   // GBK_TO_UNICODE[14568] := 16#AD6F;
   // GBK_TO_UNICODE[14569] := 16#74B7;
   // GBK_TO_UNICODE[14570] := 16#AD70;
   // GBK_TO_UNICODE[14571] := 16#74B8;
   // GBK_TO_UNICODE[14572] := 16#AD71;
   // GBK_TO_UNICODE[14573] := 16#74B9;
   // GBK_TO_UNICODE[14574] := 16#AD72;
   // GBK_TO_UNICODE[14575] := 16#74BB;
   // GBK_TO_UNICODE[14576] := 16#AD73;
   // GBK_TO_UNICODE[14577] := 16#74BC;
   // GBK_TO_UNICODE[14578] := 16#AD74;
   // GBK_TO_UNICODE[14579] := 16#74BD;
   // GBK_TO_UNICODE[14580] := 16#AD75;
   // GBK_TO_UNICODE[14581] := 16#74BE;
   // GBK_TO_UNICODE[14582] := 16#AD76;
   // GBK_TO_UNICODE[14583] := 16#74BF;
   // GBK_TO_UNICODE[14584] := 16#AD77;
   // GBK_TO_UNICODE[14585] := 16#74C0;
   // GBK_TO_UNICODE[14586] := 16#AD78;
   // GBK_TO_UNICODE[14587] := 16#74C1;
   // GBK_TO_UNICODE[14588] := 16#AD79;
   // GBK_TO_UNICODE[14589] := 16#74C2;
   // GBK_TO_UNICODE[14590] := 16#AD7A;
   // GBK_TO_UNICODE[14591] := 16#74C3;
   // GBK_TO_UNICODE[14592] := 16#AD7B;
   // GBK_TO_UNICODE[14593] := 16#74C4;
   // GBK_TO_UNICODE[14594] := 16#AD7C;
   // GBK_TO_UNICODE[14595] := 16#74C5;
   // GBK_TO_UNICODE[14596] := 16#AD7D;
   // GBK_TO_UNICODE[14597] := 16#74C6;
   // GBK_TO_UNICODE[14598] := 16#AD7E;
   // GBK_TO_UNICODE[14599] := 16#74C7;
   // GBK_TO_UNICODE[14600] := 16#AD80;
   // GBK_TO_UNICODE[14601] := 16#74C8;
   // GBK_TO_UNICODE[14602] := 16#AD81;
   // GBK_TO_UNICODE[14603] := 16#74C9;
   // GBK_TO_UNICODE[14604] := 16#AD82;
   // GBK_TO_UNICODE[14605] := 16#74CA;
   // GBK_TO_UNICODE[14606] := 16#AD83;
   // GBK_TO_UNICODE[14607] := 16#74CB;
   // GBK_TO_UNICODE[14608] := 16#AD84;
   // GBK_TO_UNICODE[14609] := 16#74CC;
   // GBK_TO_UNICODE[14610] := 16#AD85;
   // GBK_TO_UNICODE[14611] := 16#74CD;
   // GBK_TO_UNICODE[14612] := 16#AD86;
   // GBK_TO_UNICODE[14613] := 16#74CE;
   // GBK_TO_UNICODE[14614] := 16#AD87;
   // GBK_TO_UNICODE[14615] := 16#74CF;
   // GBK_TO_UNICODE[14616] := 16#AD88;
   // GBK_TO_UNICODE[14617] := 16#74D0;
   // GBK_TO_UNICODE[14618] := 16#AD89;
   // GBK_TO_UNICODE[14619] := 16#74D1;
   // GBK_TO_UNICODE[14620] := 16#AD8A;
   // GBK_TO_UNICODE[14621] := 16#74D3;
   // GBK_TO_UNICODE[14622] := 16#AD8B;
   // GBK_TO_UNICODE[14623] := 16#74D4;
   // GBK_TO_UNICODE[14624] := 16#AD8C;
   // GBK_TO_UNICODE[14625] := 16#74D5;
   // GBK_TO_UNICODE[14626] := 16#AD8D;
   // GBK_TO_UNICODE[14627] := 16#74D6;
   // GBK_TO_UNICODE[14628] := 16#AD8E;
   // GBK_TO_UNICODE[14629] := 16#74D7;
   // GBK_TO_UNICODE[14630] := 16#AD8F;
   // GBK_TO_UNICODE[14631] := 16#74D8;
   // GBK_TO_UNICODE[14632] := 16#AD90;
   // GBK_TO_UNICODE[14633] := 16#74D9;
   // GBK_TO_UNICODE[14634] := 16#AD91;
   // GBK_TO_UNICODE[14635] := 16#74DA;
   // GBK_TO_UNICODE[14636] := 16#AD92;
   // GBK_TO_UNICODE[14637] := 16#74DB;
   // GBK_TO_UNICODE[14638] := 16#AD93;
   // GBK_TO_UNICODE[14639] := 16#74DD;
   // GBK_TO_UNICODE[14640] := 16#AD94;
   // GBK_TO_UNICODE[14641] := 16#74DF;
   // GBK_TO_UNICODE[14642] := 16#AD95;
   // GBK_TO_UNICODE[14643] := 16#74E1;
   // GBK_TO_UNICODE[14644] := 16#AD96;
   // GBK_TO_UNICODE[14645] := 16#74E5;
   // GBK_TO_UNICODE[14646] := 16#AD97;
   // GBK_TO_UNICODE[14647] := 16#74E7;
   // GBK_TO_UNICODE[14648] := 16#AD98;
   // GBK_TO_UNICODE[14649] := 16#74E8;
   // GBK_TO_UNICODE[14650] := 16#AD99;
   // GBK_TO_UNICODE[14651] := 16#74E9;
   // GBK_TO_UNICODE[14652] := 16#AD9A;
   // GBK_TO_UNICODE[14653] := 16#74EA;
   // GBK_TO_UNICODE[14654] := 16#AD9B;
   // GBK_TO_UNICODE[14655] := 16#74EB;
   // GBK_TO_UNICODE[14656] := 16#AD9C;
   // GBK_TO_UNICODE[14657] := 16#74EC;
   // GBK_TO_UNICODE[14658] := 16#AD9D;
   // GBK_TO_UNICODE[14659] := 16#74ED;
   // GBK_TO_UNICODE[14660] := 16#AD9E;
   // GBK_TO_UNICODE[14661] := 16#74F0;
   // GBK_TO_UNICODE[14662] := 16#AD9F;
   // GBK_TO_UNICODE[14663] := 16#74F1;
   // GBK_TO_UNICODE[14664] := 16#ADA0;
   // GBK_TO_UNICODE[14665] := 16#74F2;
   // GBK_TO_UNICODE[14666] := 16#AE40;
   // GBK_TO_UNICODE[14667] := 16#74F3;
   // GBK_TO_UNICODE[14668] := 16#AE41;
   // GBK_TO_UNICODE[14669] := 16#74F5;
   // GBK_TO_UNICODE[14670] := 16#AE42;
   // GBK_TO_UNICODE[14671] := 16#74F8;
   // GBK_TO_UNICODE[14672] := 16#AE43;
   // GBK_TO_UNICODE[14673] := 16#74F9;
   // GBK_TO_UNICODE[14674] := 16#AE44;
   // GBK_TO_UNICODE[14675] := 16#74FA;
   // GBK_TO_UNICODE[14676] := 16#AE45;
   // GBK_TO_UNICODE[14677] := 16#74FB;
   // GBK_TO_UNICODE[14678] := 16#AE46;
   // GBK_TO_UNICODE[14679] := 16#74FC;
   // GBK_TO_UNICODE[14680] := 16#AE47;
   // GBK_TO_UNICODE[14681] := 16#74FD;
   // GBK_TO_UNICODE[14682] := 16#AE48;
   // GBK_TO_UNICODE[14683] := 16#74FE;
   // GBK_TO_UNICODE[14684] := 16#AE49;
   // GBK_TO_UNICODE[14685] := 16#7500;
   // GBK_TO_UNICODE[14686] := 16#AE4A;
   // GBK_TO_UNICODE[14687] := 16#7501;
   // GBK_TO_UNICODE[14688] := 16#AE4B;
   // GBK_TO_UNICODE[14689] := 16#7502;
   // GBK_TO_UNICODE[14690] := 16#AE4C;
   // GBK_TO_UNICODE[14691] := 16#7503;
   // GBK_TO_UNICODE[14692] := 16#AE4D;
   // GBK_TO_UNICODE[14693] := 16#7505;
   // GBK_TO_UNICODE[14694] := 16#AE4E;
   // GBK_TO_UNICODE[14695] := 16#7506;
   // GBK_TO_UNICODE[14696] := 16#AE4F;
   // GBK_TO_UNICODE[14697] := 16#7507;
   // GBK_TO_UNICODE[14698] := 16#AE50;
   // GBK_TO_UNICODE[14699] := 16#7508;
   // GBK_TO_UNICODE[14700] := 16#AE51;
   // GBK_TO_UNICODE[14701] := 16#7509;
   // GBK_TO_UNICODE[14702] := 16#AE52;
   // GBK_TO_UNICODE[14703] := 16#750A;
   // GBK_TO_UNICODE[14704] := 16#AE53;
   // GBK_TO_UNICODE[14705] := 16#750B;
   // GBK_TO_UNICODE[14706] := 16#AE54;
   // GBK_TO_UNICODE[14707] := 16#750C;
   // GBK_TO_UNICODE[14708] := 16#AE55;
   // GBK_TO_UNICODE[14709] := 16#750E;
   // GBK_TO_UNICODE[14710] := 16#AE56;
   // GBK_TO_UNICODE[14711] := 16#7510;
   // GBK_TO_UNICODE[14712] := 16#AE57;
   // GBK_TO_UNICODE[14713] := 16#7512;
   // GBK_TO_UNICODE[14714] := 16#AE58;
   // GBK_TO_UNICODE[14715] := 16#7514;
   // GBK_TO_UNICODE[14716] := 16#AE59;
   // GBK_TO_UNICODE[14717] := 16#7515;
   // GBK_TO_UNICODE[14718] := 16#AE5A;
   // GBK_TO_UNICODE[14719] := 16#7516;
   // GBK_TO_UNICODE[14720] := 16#AE5B;
   // GBK_TO_UNICODE[14721] := 16#7517;
   // GBK_TO_UNICODE[14722] := 16#AE5C;
   // GBK_TO_UNICODE[14723] := 16#751B;
   // GBK_TO_UNICODE[14724] := 16#AE5D;
   // GBK_TO_UNICODE[14725] := 16#751D;
   // GBK_TO_UNICODE[14726] := 16#AE5E;
   // GBK_TO_UNICODE[14727] := 16#751E;
   // GBK_TO_UNICODE[14728] := 16#AE5F;
   // GBK_TO_UNICODE[14729] := 16#7520;
   // GBK_TO_UNICODE[14730] := 16#AE60;
   // GBK_TO_UNICODE[14731] := 16#7521;
   // GBK_TO_UNICODE[14732] := 16#AE61;
   // GBK_TO_UNICODE[14733] := 16#7522;
   // GBK_TO_UNICODE[14734] := 16#AE62;
   // GBK_TO_UNICODE[14735] := 16#7523;
   // GBK_TO_UNICODE[14736] := 16#AE63;
   // GBK_TO_UNICODE[14737] := 16#7524;
   // GBK_TO_UNICODE[14738] := 16#AE64;
   // GBK_TO_UNICODE[14739] := 16#7526;
   // GBK_TO_UNICODE[14740] := 16#AE65;
   // GBK_TO_UNICODE[14741] := 16#7527;
   // GBK_TO_UNICODE[14742] := 16#AE66;
   // GBK_TO_UNICODE[14743] := 16#752A;
   // GBK_TO_UNICODE[14744] := 16#AE67;
   // GBK_TO_UNICODE[14745] := 16#752E;
   // GBK_TO_UNICODE[14746] := 16#AE68;
   // GBK_TO_UNICODE[14747] := 16#7534;
   // GBK_TO_UNICODE[14748] := 16#AE69;
   // GBK_TO_UNICODE[14749] := 16#7536;
   // GBK_TO_UNICODE[14750] := 16#AE6A;
   // GBK_TO_UNICODE[14751] := 16#7539;
   // GBK_TO_UNICODE[14752] := 16#AE6B;
   // GBK_TO_UNICODE[14753] := 16#753C;
   // GBK_TO_UNICODE[14754] := 16#AE6C;
   // GBK_TO_UNICODE[14755] := 16#753D;
   // GBK_TO_UNICODE[14756] := 16#AE6D;
   // GBK_TO_UNICODE[14757] := 16#753F;
   // GBK_TO_UNICODE[14758] := 16#AE6E;
   // GBK_TO_UNICODE[14759] := 16#7541;
   // GBK_TO_UNICODE[14760] := 16#AE6F;
   // GBK_TO_UNICODE[14761] := 16#7542;
   // GBK_TO_UNICODE[14762] := 16#AE70;
   // GBK_TO_UNICODE[14763] := 16#7543;
   // GBK_TO_UNICODE[14764] := 16#AE71;
   // GBK_TO_UNICODE[14765] := 16#7544;
   // GBK_TO_UNICODE[14766] := 16#AE72;
   // GBK_TO_UNICODE[14767] := 16#7546;
   // GBK_TO_UNICODE[14768] := 16#AE73;
   // GBK_TO_UNICODE[14769] := 16#7547;
   // GBK_TO_UNICODE[14770] := 16#AE74;
   // GBK_TO_UNICODE[14771] := 16#7549;
   // GBK_TO_UNICODE[14772] := 16#AE75;
   // GBK_TO_UNICODE[14773] := 16#754A;
   // GBK_TO_UNICODE[14774] := 16#AE76;
   // GBK_TO_UNICODE[14775] := 16#754D;
   // GBK_TO_UNICODE[14776] := 16#AE77;
   // GBK_TO_UNICODE[14777] := 16#7550;
   // GBK_TO_UNICODE[14778] := 16#AE78;
   // GBK_TO_UNICODE[14779] := 16#7551;
   // GBK_TO_UNICODE[14780] := 16#AE79;
   // GBK_TO_UNICODE[14781] := 16#7552;
   // GBK_TO_UNICODE[14782] := 16#AE7A;
   // GBK_TO_UNICODE[14783] := 16#7553;
   // GBK_TO_UNICODE[14784] := 16#AE7B;
   // GBK_TO_UNICODE[14785] := 16#7555;
   // GBK_TO_UNICODE[14786] := 16#AE7C;
   // GBK_TO_UNICODE[14787] := 16#7556;
   // GBK_TO_UNICODE[14788] := 16#AE7D;
   // GBK_TO_UNICODE[14789] := 16#7557;
   // GBK_TO_UNICODE[14790] := 16#AE7E;
   // GBK_TO_UNICODE[14791] := 16#7558;
   // GBK_TO_UNICODE[14792] := 16#AE80;
   // GBK_TO_UNICODE[14793] := 16#755D;
   // GBK_TO_UNICODE[14794] := 16#AE81;
   // GBK_TO_UNICODE[14795] := 16#755E;
   // GBK_TO_UNICODE[14796] := 16#AE82;
   // GBK_TO_UNICODE[14797] := 16#755F;
   // GBK_TO_UNICODE[14798] := 16#AE83;
   // GBK_TO_UNICODE[14799] := 16#7560;
   // GBK_TO_UNICODE[14800] := 16#AE84;
   // GBK_TO_UNICODE[14801] := 16#7561;
   // GBK_TO_UNICODE[14802] := 16#AE85;
   // GBK_TO_UNICODE[14803] := 16#7562;
   // GBK_TO_UNICODE[14804] := 16#AE86;
   // GBK_TO_UNICODE[14805] := 16#7563;
   // GBK_TO_UNICODE[14806] := 16#AE87;
   // GBK_TO_UNICODE[14807] := 16#7564;
   // GBK_TO_UNICODE[14808] := 16#AE88;
   // GBK_TO_UNICODE[14809] := 16#7567;
   // GBK_TO_UNICODE[14810] := 16#AE89;
   // GBK_TO_UNICODE[14811] := 16#7568;
   // GBK_TO_UNICODE[14812] := 16#AE8A;
   // GBK_TO_UNICODE[14813] := 16#7569;
   // GBK_TO_UNICODE[14814] := 16#AE8B;
   // GBK_TO_UNICODE[14815] := 16#756B;
   // GBK_TO_UNICODE[14816] := 16#AE8C;
   // GBK_TO_UNICODE[14817] := 16#756C;
   // GBK_TO_UNICODE[14818] := 16#AE8D;
   // GBK_TO_UNICODE[14819] := 16#756D;
   // GBK_TO_UNICODE[14820] := 16#AE8E;
   // GBK_TO_UNICODE[14821] := 16#756E;
   // GBK_TO_UNICODE[14822] := 16#AE8F;
   // GBK_TO_UNICODE[14823] := 16#756F;
   // GBK_TO_UNICODE[14824] := 16#AE90;
   // GBK_TO_UNICODE[14825] := 16#7570;
   // GBK_TO_UNICODE[14826] := 16#AE91;
   // GBK_TO_UNICODE[14827] := 16#7571;
   // GBK_TO_UNICODE[14828] := 16#AE92;
   // GBK_TO_UNICODE[14829] := 16#7573;
   // GBK_TO_UNICODE[14830] := 16#AE93;
   // GBK_TO_UNICODE[14831] := 16#7575;
   // GBK_TO_UNICODE[14832] := 16#AE94;
   // GBK_TO_UNICODE[14833] := 16#7576;
   // GBK_TO_UNICODE[14834] := 16#AE95;
   // GBK_TO_UNICODE[14835] := 16#7577;
   // GBK_TO_UNICODE[14836] := 16#AE96;
   // GBK_TO_UNICODE[14837] := 16#757A;
   // GBK_TO_UNICODE[14838] := 16#AE97;
   // GBK_TO_UNICODE[14839] := 16#757B;
   // GBK_TO_UNICODE[14840] := 16#AE98;
   // GBK_TO_UNICODE[14841] := 16#757C;
   // GBK_TO_UNICODE[14842] := 16#AE99;
   // GBK_TO_UNICODE[14843] := 16#757D;
   // GBK_TO_UNICODE[14844] := 16#AE9A;
   // GBK_TO_UNICODE[14845] := 16#757E;
   // GBK_TO_UNICODE[14846] := 16#AE9B;
   // GBK_TO_UNICODE[14847] := 16#7580;
   // GBK_TO_UNICODE[14848] := 16#AE9C;
   // GBK_TO_UNICODE[14849] := 16#7581;
   // GBK_TO_UNICODE[14850] := 16#AE9D;
   // GBK_TO_UNICODE[14851] := 16#7582;
   // GBK_TO_UNICODE[14852] := 16#AE9E;
   // GBK_TO_UNICODE[14853] := 16#7584;
   // GBK_TO_UNICODE[14854] := 16#AE9F;
   // GBK_TO_UNICODE[14855] := 16#7585;
   // GBK_TO_UNICODE[14856] := 16#AEA0;
   // GBK_TO_UNICODE[14857] := 16#7587;
   // GBK_TO_UNICODE[14858] := 16#AF40;
   // GBK_TO_UNICODE[14859] := 16#7588;
   // GBK_TO_UNICODE[14860] := 16#AF41;
   // GBK_TO_UNICODE[14861] := 16#7589;
   // GBK_TO_UNICODE[14862] := 16#AF42;
   // GBK_TO_UNICODE[14863] := 16#758A;
   // GBK_TO_UNICODE[14864] := 16#AF43;
   // GBK_TO_UNICODE[14865] := 16#758C;
   // GBK_TO_UNICODE[14866] := 16#AF44;
   // GBK_TO_UNICODE[14867] := 16#758D;
   // GBK_TO_UNICODE[14868] := 16#AF45;
   // GBK_TO_UNICODE[14869] := 16#758E;
   // GBK_TO_UNICODE[14870] := 16#AF46;
   // GBK_TO_UNICODE[14871] := 16#7590;
   // GBK_TO_UNICODE[14872] := 16#AF47;
   // GBK_TO_UNICODE[14873] := 16#7593;
   // GBK_TO_UNICODE[14874] := 16#AF48;
   // GBK_TO_UNICODE[14875] := 16#7595;
   // GBK_TO_UNICODE[14876] := 16#AF49;
   // GBK_TO_UNICODE[14877] := 16#7598;
   // GBK_TO_UNICODE[14878] := 16#AF4A;
   // GBK_TO_UNICODE[14879] := 16#759B;
   // GBK_TO_UNICODE[14880] := 16#AF4B;
   // GBK_TO_UNICODE[14881] := 16#759C;
   // GBK_TO_UNICODE[14882] := 16#AF4C;
   // GBK_TO_UNICODE[14883] := 16#759E;
   // GBK_TO_UNICODE[14884] := 16#AF4D;
   // GBK_TO_UNICODE[14885] := 16#75A2;
   // GBK_TO_UNICODE[14886] := 16#AF4E;
   // GBK_TO_UNICODE[14887] := 16#75A6;
   // GBK_TO_UNICODE[14888] := 16#AF4F;
   // GBK_TO_UNICODE[14889] := 16#75A7;
   // GBK_TO_UNICODE[14890] := 16#AF50;
   // GBK_TO_UNICODE[14891] := 16#75A8;
   // GBK_TO_UNICODE[14892] := 16#AF51;
   // GBK_TO_UNICODE[14893] := 16#75A9;
   // GBK_TO_UNICODE[14894] := 16#AF52;
   // GBK_TO_UNICODE[14895] := 16#75AA;
   // GBK_TO_UNICODE[14896] := 16#AF53;
   // GBK_TO_UNICODE[14897] := 16#75AD;
   // GBK_TO_UNICODE[14898] := 16#AF54;
   // GBK_TO_UNICODE[14899] := 16#75B6;
   // GBK_TO_UNICODE[14900] := 16#AF55;
   // GBK_TO_UNICODE[14901] := 16#75B7;
   // GBK_TO_UNICODE[14902] := 16#AF56;
   // GBK_TO_UNICODE[14903] := 16#75BA;
   // GBK_TO_UNICODE[14904] := 16#AF57;
   // GBK_TO_UNICODE[14905] := 16#75BB;
   // GBK_TO_UNICODE[14906] := 16#AF58;
   // GBK_TO_UNICODE[14907] := 16#75BF;
   // GBK_TO_UNICODE[14908] := 16#AF59;
   // GBK_TO_UNICODE[14909] := 16#75C0;
   // GBK_TO_UNICODE[14910] := 16#AF5A;
   // GBK_TO_UNICODE[14911] := 16#75C1;
   // GBK_TO_UNICODE[14912] := 16#AF5B;
   // GBK_TO_UNICODE[14913] := 16#75C6;
   // GBK_TO_UNICODE[14914] := 16#AF5C;
   // GBK_TO_UNICODE[14915] := 16#75CB;
   // GBK_TO_UNICODE[14916] := 16#AF5D;
   // GBK_TO_UNICODE[14917] := 16#75CC;
   // GBK_TO_UNICODE[14918] := 16#AF5E;
   // GBK_TO_UNICODE[14919] := 16#75CE;
   // GBK_TO_UNICODE[14920] := 16#AF5F;
   // GBK_TO_UNICODE[14921] := 16#75CF;
   // GBK_TO_UNICODE[14922] := 16#AF60;
   // GBK_TO_UNICODE[14923] := 16#75D0;
   // GBK_TO_UNICODE[14924] := 16#AF61;
   // GBK_TO_UNICODE[14925] := 16#75D1;
   // GBK_TO_UNICODE[14926] := 16#AF62;
   // GBK_TO_UNICODE[14927] := 16#75D3;
   // GBK_TO_UNICODE[14928] := 16#AF63;
   // GBK_TO_UNICODE[14929] := 16#75D7;
   // GBK_TO_UNICODE[14930] := 16#AF64;
   // GBK_TO_UNICODE[14931] := 16#75D9;
   // GBK_TO_UNICODE[14932] := 16#AF65;
   // GBK_TO_UNICODE[14933] := 16#75DA;
   // GBK_TO_UNICODE[14934] := 16#AF66;
   // GBK_TO_UNICODE[14935] := 16#75DC;
   // GBK_TO_UNICODE[14936] := 16#AF67;
   // GBK_TO_UNICODE[14937] := 16#75DD;
   // GBK_TO_UNICODE[14938] := 16#AF68;
   // GBK_TO_UNICODE[14939] := 16#75DF;
   // GBK_TO_UNICODE[14940] := 16#AF69;
   // GBK_TO_UNICODE[14941] := 16#75E0;
   // GBK_TO_UNICODE[14942] := 16#AF6A;
   // GBK_TO_UNICODE[14943] := 16#75E1;
   // GBK_TO_UNICODE[14944] := 16#AF6B;
   // GBK_TO_UNICODE[14945] := 16#75E5;
   // GBK_TO_UNICODE[14946] := 16#AF6C;
   // GBK_TO_UNICODE[14947] := 16#75E9;
   // GBK_TO_UNICODE[14948] := 16#AF6D;
   // GBK_TO_UNICODE[14949] := 16#75EC;
   // GBK_TO_UNICODE[14950] := 16#AF6E;
   // GBK_TO_UNICODE[14951] := 16#75ED;
   // GBK_TO_UNICODE[14952] := 16#AF6F;
   // GBK_TO_UNICODE[14953] := 16#75EE;
   // GBK_TO_UNICODE[14954] := 16#AF70;
   // GBK_TO_UNICODE[14955] := 16#75EF;
   // GBK_TO_UNICODE[14956] := 16#AF71;
   // GBK_TO_UNICODE[14957] := 16#75F2;
   // GBK_TO_UNICODE[14958] := 16#AF72;
   // GBK_TO_UNICODE[14959] := 16#75F3;
   // GBK_TO_UNICODE[14960] := 16#AF73;
   // GBK_TO_UNICODE[14961] := 16#75F5;
   // GBK_TO_UNICODE[14962] := 16#AF74;
   // GBK_TO_UNICODE[14963] := 16#75F6;
   // GBK_TO_UNICODE[14964] := 16#AF75;
   // GBK_TO_UNICODE[14965] := 16#75F7;
   // GBK_TO_UNICODE[14966] := 16#AF76;
   // GBK_TO_UNICODE[14967] := 16#75F8;
   // GBK_TO_UNICODE[14968] := 16#AF77;
   // GBK_TO_UNICODE[14969] := 16#75FA;
   // GBK_TO_UNICODE[14970] := 16#AF78;
   // GBK_TO_UNICODE[14971] := 16#75FB;
   // GBK_TO_UNICODE[14972] := 16#AF79;
   // GBK_TO_UNICODE[14973] := 16#75FD;
   // GBK_TO_UNICODE[14974] := 16#AF7A;
   // GBK_TO_UNICODE[14975] := 16#75FE;
   // GBK_TO_UNICODE[14976] := 16#AF7B;
   // GBK_TO_UNICODE[14977] := 16#7602;
   // GBK_TO_UNICODE[14978] := 16#AF7C;
   // GBK_TO_UNICODE[14979] := 16#7604;
   // GBK_TO_UNICODE[14980] := 16#AF7D;
   // GBK_TO_UNICODE[14981] := 16#7606;
   // GBK_TO_UNICODE[14982] := 16#AF7E;
   // GBK_TO_UNICODE[14983] := 16#7607;
   // GBK_TO_UNICODE[14984] := 16#AF80;
   // GBK_TO_UNICODE[14985] := 16#7608;
   // GBK_TO_UNICODE[14986] := 16#AF81;
   // GBK_TO_UNICODE[14987] := 16#7609;
   // GBK_TO_UNICODE[14988] := 16#AF82;
   // GBK_TO_UNICODE[14989] := 16#760B;
   // GBK_TO_UNICODE[14990] := 16#AF83;
   // GBK_TO_UNICODE[14991] := 16#760D;
   // GBK_TO_UNICODE[14992] := 16#AF84;
   // GBK_TO_UNICODE[14993] := 16#760E;
   // GBK_TO_UNICODE[14994] := 16#AF85;
   // GBK_TO_UNICODE[14995] := 16#760F;
   // GBK_TO_UNICODE[14996] := 16#AF86;
   // GBK_TO_UNICODE[14997] := 16#7611;
   // GBK_TO_UNICODE[14998] := 16#AF87;
   // GBK_TO_UNICODE[14999] := 16#7612;
   // GBK_TO_UNICODE[15000] := 16#AF88;
   // GBK_TO_UNICODE[15001] := 16#7613;
   // GBK_TO_UNICODE[15002] := 16#AF89;
   // GBK_TO_UNICODE[15003] := 16#7614;
   // GBK_TO_UNICODE[15004] := 16#AF8A;
   // GBK_TO_UNICODE[15005] := 16#7616;
   // GBK_TO_UNICODE[15006] := 16#AF8B;
   // GBK_TO_UNICODE[15007] := 16#761A;
   // GBK_TO_UNICODE[15008] := 16#AF8C;
   // GBK_TO_UNICODE[15009] := 16#761C;
   // GBK_TO_UNICODE[15010] := 16#AF8D;
   // GBK_TO_UNICODE[15011] := 16#761D;
   // GBK_TO_UNICODE[15012] := 16#AF8E;
   // GBK_TO_UNICODE[15013] := 16#761E;
   // GBK_TO_UNICODE[15014] := 16#AF8F;
   // GBK_TO_UNICODE[15015] := 16#7621;
   // GBK_TO_UNICODE[15016] := 16#AF90;
   // GBK_TO_UNICODE[15017] := 16#7623;
   // GBK_TO_UNICODE[15018] := 16#AF91;
   // GBK_TO_UNICODE[15019] := 16#7627;
   // GBK_TO_UNICODE[15020] := 16#AF92;
   // GBK_TO_UNICODE[15021] := 16#7628;
   // GBK_TO_UNICODE[15022] := 16#AF93;
   // GBK_TO_UNICODE[15023] := 16#762C;
   // GBK_TO_UNICODE[15024] := 16#AF94;
   // GBK_TO_UNICODE[15025] := 16#762E;
   // GBK_TO_UNICODE[15026] := 16#AF95;
   // GBK_TO_UNICODE[15027] := 16#762F;
   // GBK_TO_UNICODE[15028] := 16#AF96;
   // GBK_TO_UNICODE[15029] := 16#7631;
   // GBK_TO_UNICODE[15030] := 16#AF97;
   // GBK_TO_UNICODE[15031] := 16#7632;
   // GBK_TO_UNICODE[15032] := 16#AF98;
   // GBK_TO_UNICODE[15033] := 16#7636;
   // GBK_TO_UNICODE[15034] := 16#AF99;
   // GBK_TO_UNICODE[15035] := 16#7637;
   // GBK_TO_UNICODE[15036] := 16#AF9A;
   // GBK_TO_UNICODE[15037] := 16#7639;
   // GBK_TO_UNICODE[15038] := 16#AF9B;
   // GBK_TO_UNICODE[15039] := 16#763A;
   // GBK_TO_UNICODE[15040] := 16#AF9C;
   // GBK_TO_UNICODE[15041] := 16#763B;
   // GBK_TO_UNICODE[15042] := 16#AF9D;
   // GBK_TO_UNICODE[15043] := 16#763D;
   // GBK_TO_UNICODE[15044] := 16#AF9E;
   // GBK_TO_UNICODE[15045] := 16#7641;
   // GBK_TO_UNICODE[15046] := 16#AF9F;
   // GBK_TO_UNICODE[15047] := 16#7642;
   // GBK_TO_UNICODE[15048] := 16#AFA0;
   // GBK_TO_UNICODE[15049] := 16#7644;
   // GBK_TO_UNICODE[15050] := 16#B040;
   // GBK_TO_UNICODE[15051] := 16#7645;
   // GBK_TO_UNICODE[15052] := 16#B041;
   // GBK_TO_UNICODE[15053] := 16#7646;
   // GBK_TO_UNICODE[15054] := 16#B042;
   // GBK_TO_UNICODE[15055] := 16#7647;
   // GBK_TO_UNICODE[15056] := 16#B043;
   // GBK_TO_UNICODE[15057] := 16#7648;
   // GBK_TO_UNICODE[15058] := 16#B044;
   // GBK_TO_UNICODE[15059] := 16#7649;
   // GBK_TO_UNICODE[15060] := 16#B045;
   // GBK_TO_UNICODE[15061] := 16#764A;
   // GBK_TO_UNICODE[15062] := 16#B046;
   // GBK_TO_UNICODE[15063] := 16#764B;
   // GBK_TO_UNICODE[15064] := 16#B047;
   // GBK_TO_UNICODE[15065] := 16#764E;
   // GBK_TO_UNICODE[15066] := 16#B048;
   // GBK_TO_UNICODE[15067] := 16#764F;
   // GBK_TO_UNICODE[15068] := 16#B049;
   // GBK_TO_UNICODE[15069] := 16#7650;
   // GBK_TO_UNICODE[15070] := 16#B04A;
   // GBK_TO_UNICODE[15071] := 16#7651;
   // GBK_TO_UNICODE[15072] := 16#B04B;
   // GBK_TO_UNICODE[15073] := 16#7652;
   // GBK_TO_UNICODE[15074] := 16#B04C;
   // GBK_TO_UNICODE[15075] := 16#7653;
   // GBK_TO_UNICODE[15076] := 16#B04D;
   // GBK_TO_UNICODE[15077] := 16#7655;
   // GBK_TO_UNICODE[15078] := 16#B04E;
   // GBK_TO_UNICODE[15079] := 16#7657;
   // GBK_TO_UNICODE[15080] := 16#B04F;
   // GBK_TO_UNICODE[15081] := 16#7658;
   // GBK_TO_UNICODE[15082] := 16#B050;
   // GBK_TO_UNICODE[15083] := 16#7659;
   // GBK_TO_UNICODE[15084] := 16#B051;
   // GBK_TO_UNICODE[15085] := 16#765A;
   // GBK_TO_UNICODE[15086] := 16#B052;
   // GBK_TO_UNICODE[15087] := 16#765B;
   // GBK_TO_UNICODE[15088] := 16#B053;
   // GBK_TO_UNICODE[15089] := 16#765D;
   // GBK_TO_UNICODE[15090] := 16#B054;
   // GBK_TO_UNICODE[15091] := 16#765F;
   // GBK_TO_UNICODE[15092] := 16#B055;
   // GBK_TO_UNICODE[15093] := 16#7660;
   // GBK_TO_UNICODE[15094] := 16#B056;
   // GBK_TO_UNICODE[15095] := 16#7661;
   // GBK_TO_UNICODE[15096] := 16#B057;
   // GBK_TO_UNICODE[15097] := 16#7662;
   // GBK_TO_UNICODE[15098] := 16#B058;
   // GBK_TO_UNICODE[15099] := 16#7664;
   // GBK_TO_UNICODE[15100] := 16#B059;
   // GBK_TO_UNICODE[15101] := 16#7665;
   // GBK_TO_UNICODE[15102] := 16#B05A;
   // GBK_TO_UNICODE[15103] := 16#7666;
   // GBK_TO_UNICODE[15104] := 16#B05B;
   // GBK_TO_UNICODE[15105] := 16#7667;
   // GBK_TO_UNICODE[15106] := 16#B05C;
   // GBK_TO_UNICODE[15107] := 16#7668;
   // GBK_TO_UNICODE[15108] := 16#B05D;
   // GBK_TO_UNICODE[15109] := 16#7669;
   // GBK_TO_UNICODE[15110] := 16#B05E;
   // GBK_TO_UNICODE[15111] := 16#766A;
   // GBK_TO_UNICODE[15112] := 16#B05F;
   // GBK_TO_UNICODE[15113] := 16#766C;
   // GBK_TO_UNICODE[15114] := 16#B060;
   // GBK_TO_UNICODE[15115] := 16#766D;
   // GBK_TO_UNICODE[15116] := 16#B061;
   // GBK_TO_UNICODE[15117] := 16#766E;
   // GBK_TO_UNICODE[15118] := 16#B062;
   // GBK_TO_UNICODE[15119] := 16#7670;
   // GBK_TO_UNICODE[15120] := 16#B063;
   // GBK_TO_UNICODE[15121] := 16#7671;
   // GBK_TO_UNICODE[15122] := 16#B064;
   // GBK_TO_UNICODE[15123] := 16#7672;
   // GBK_TO_UNICODE[15124] := 16#B065;
   // GBK_TO_UNICODE[15125] := 16#7673;
   // GBK_TO_UNICODE[15126] := 16#B066;
   // GBK_TO_UNICODE[15127] := 16#7674;
   // GBK_TO_UNICODE[15128] := 16#B067;
   // GBK_TO_UNICODE[15129] := 16#7675;
   // GBK_TO_UNICODE[15130] := 16#B068;
   // GBK_TO_UNICODE[15131] := 16#7676;
   // GBK_TO_UNICODE[15132] := 16#B069;
   // GBK_TO_UNICODE[15133] := 16#7677;
   // GBK_TO_UNICODE[15134] := 16#B06A;
   // GBK_TO_UNICODE[15135] := 16#7679;
   // GBK_TO_UNICODE[15136] := 16#B06B;
   // GBK_TO_UNICODE[15137] := 16#767A;
   // GBK_TO_UNICODE[15138] := 16#B06C;
   // GBK_TO_UNICODE[15139] := 16#767C;
   // GBK_TO_UNICODE[15140] := 16#B06D;
   // GBK_TO_UNICODE[15141] := 16#767F;
   // GBK_TO_UNICODE[15142] := 16#B06E;
   // GBK_TO_UNICODE[15143] := 16#7680;
   // GBK_TO_UNICODE[15144] := 16#B06F;
   // GBK_TO_UNICODE[15145] := 16#7681;
   // GBK_TO_UNICODE[15146] := 16#B070;
   // GBK_TO_UNICODE[15147] := 16#7683;
   // GBK_TO_UNICODE[15148] := 16#B071;
   // GBK_TO_UNICODE[15149] := 16#7685;
   // GBK_TO_UNICODE[15150] := 16#B072;
   // GBK_TO_UNICODE[15151] := 16#7689;
   // GBK_TO_UNICODE[15152] := 16#B073;
   // GBK_TO_UNICODE[15153] := 16#768A;
   // GBK_TO_UNICODE[15154] := 16#B074;
   // GBK_TO_UNICODE[15155] := 16#768C;
   // GBK_TO_UNICODE[15156] := 16#B075;
   // GBK_TO_UNICODE[15157] := 16#768D;
   // GBK_TO_UNICODE[15158] := 16#B076;
   // GBK_TO_UNICODE[15159] := 16#768F;
   // GBK_TO_UNICODE[15160] := 16#B077;
   // GBK_TO_UNICODE[15161] := 16#7690;
   // GBK_TO_UNICODE[15162] := 16#B078;
   // GBK_TO_UNICODE[15163] := 16#7692;
   // GBK_TO_UNICODE[15164] := 16#B079;
   // GBK_TO_UNICODE[15165] := 16#7694;
   // GBK_TO_UNICODE[15166] := 16#B07A;
   // GBK_TO_UNICODE[15167] := 16#7695;
   // GBK_TO_UNICODE[15168] := 16#B07B;
   // GBK_TO_UNICODE[15169] := 16#7697;
   // GBK_TO_UNICODE[15170] := 16#B07C;
   // GBK_TO_UNICODE[15171] := 16#7698;
   // GBK_TO_UNICODE[15172] := 16#B07D;
   // GBK_TO_UNICODE[15173] := 16#769A;
   // GBK_TO_UNICODE[15174] := 16#B07E;
   // GBK_TO_UNICODE[15175] := 16#769B;
   // GBK_TO_UNICODE[15176] := 16#B080;
   // GBK_TO_UNICODE[15177] := 16#769C;
   // GBK_TO_UNICODE[15178] := 16#B081;
   // GBK_TO_UNICODE[15179] := 16#769D;
   // GBK_TO_UNICODE[15180] := 16#B082;
   // GBK_TO_UNICODE[15181] := 16#769E;
   // GBK_TO_UNICODE[15182] := 16#B083;
   // GBK_TO_UNICODE[15183] := 16#769F;
   // GBK_TO_UNICODE[15184] := 16#B084;
   // GBK_TO_UNICODE[15185] := 16#76A0;
   // GBK_TO_UNICODE[15186] := 16#B085;
   // GBK_TO_UNICODE[15187] := 16#76A1;
   // GBK_TO_UNICODE[15188] := 16#B086;
   // GBK_TO_UNICODE[15189] := 16#76A2;
   // GBK_TO_UNICODE[15190] := 16#B087;
   // GBK_TO_UNICODE[15191] := 16#76A3;
   // GBK_TO_UNICODE[15192] := 16#B088;
   // GBK_TO_UNICODE[15193] := 16#76A5;
   // GBK_TO_UNICODE[15194] := 16#B089;
   // GBK_TO_UNICODE[15195] := 16#76A6;
   // GBK_TO_UNICODE[15196] := 16#B08A;
   // GBK_TO_UNICODE[15197] := 16#76A7;
   // GBK_TO_UNICODE[15198] := 16#B08B;
   // GBK_TO_UNICODE[15199] := 16#76A8;
   // GBK_TO_UNICODE[15200] := 16#B08C;
   // GBK_TO_UNICODE[15201] := 16#76A9;
   // GBK_TO_UNICODE[15202] := 16#B08D;
   // GBK_TO_UNICODE[15203] := 16#76AA;
   // GBK_TO_UNICODE[15204] := 16#B08E;
   // GBK_TO_UNICODE[15205] := 16#76AB;
   // GBK_TO_UNICODE[15206] := 16#B08F;
   // GBK_TO_UNICODE[15207] := 16#76AC;
   // GBK_TO_UNICODE[15208] := 16#B090;
   // GBK_TO_UNICODE[15209] := 16#76AD;
   // GBK_TO_UNICODE[15210] := 16#B091;
   // GBK_TO_UNICODE[15211] := 16#76AF;
   // GBK_TO_UNICODE[15212] := 16#B092;
   // GBK_TO_UNICODE[15213] := 16#76B0;
   // GBK_TO_UNICODE[15214] := 16#B093;
   // GBK_TO_UNICODE[15215] := 16#76B3;
   // GBK_TO_UNICODE[15216] := 16#B094;
   // GBK_TO_UNICODE[15217] := 16#76B5;
   // GBK_TO_UNICODE[15218] := 16#B095;
   // GBK_TO_UNICODE[15219] := 16#76B6;
   // GBK_TO_UNICODE[15220] := 16#B096;
   // GBK_TO_UNICODE[15221] := 16#76B7;
   // GBK_TO_UNICODE[15222] := 16#B097;
   // GBK_TO_UNICODE[15223] := 16#76B8;
   // GBK_TO_UNICODE[15224] := 16#B098;
   // GBK_TO_UNICODE[15225] := 16#76B9;
   // GBK_TO_UNICODE[15226] := 16#B099;
   // GBK_TO_UNICODE[15227] := 16#76BA;
   // GBK_TO_UNICODE[15228] := 16#B09A;
   // GBK_TO_UNICODE[15229] := 16#76BB;
   // GBK_TO_UNICODE[15230] := 16#B09B;
   // GBK_TO_UNICODE[15231] := 16#76BC;
   // GBK_TO_UNICODE[15232] := 16#B09C;
   // GBK_TO_UNICODE[15233] := 16#76BD;
   // GBK_TO_UNICODE[15234] := 16#B09D;
   // GBK_TO_UNICODE[15235] := 16#76BE;
   // GBK_TO_UNICODE[15236] := 16#B09E;
   // GBK_TO_UNICODE[15237] := 16#76C0;
   // GBK_TO_UNICODE[15238] := 16#B09F;
   // GBK_TO_UNICODE[15239] := 16#76C1;
   // GBK_TO_UNICODE[15240] := 16#B0A0;
   // GBK_TO_UNICODE[15241] := 16#76C3;
   // GBK_TO_UNICODE[15242] := 16#B0A1;
   // GBK_TO_UNICODE[15243] := 16#554A;
   // GBK_TO_UNICODE[15244] := 16#B0A2;
   // GBK_TO_UNICODE[15245] := 16#963F;
   // GBK_TO_UNICODE[15246] := 16#B0A3;
   // GBK_TO_UNICODE[15247] := 16#57C3;
   // GBK_TO_UNICODE[15248] := 16#B0A4;
   // GBK_TO_UNICODE[15249] := 16#6328;
   // GBK_TO_UNICODE[15250] := 16#B0A5;
   // GBK_TO_UNICODE[15251] := 16#54CE;
   // GBK_TO_UNICODE[15252] := 16#B0A6;
   // GBK_TO_UNICODE[15253] := 16#5509;
   // GBK_TO_UNICODE[15254] := 16#B0A7;
   // GBK_TO_UNICODE[15255] := 16#54C0;
   // GBK_TO_UNICODE[15256] := 16#B0A8;
   // GBK_TO_UNICODE[15257] := 16#7691;
   // GBK_TO_UNICODE[15258] := 16#B0A9;
   // GBK_TO_UNICODE[15259] := 16#764C;
   // GBK_TO_UNICODE[15260] := 16#B0AA;
   // GBK_TO_UNICODE[15261] := 16#853C;
   // GBK_TO_UNICODE[15262] := 16#B0AB;
   // GBK_TO_UNICODE[15263] := 16#77EE;
   // GBK_TO_UNICODE[15264] := 16#B0AC;
   // GBK_TO_UNICODE[15265] := 16#827E;
   // GBK_TO_UNICODE[15266] := 16#B0AD;
   // GBK_TO_UNICODE[15267] := 16#788D;
   // GBK_TO_UNICODE[15268] := 16#B0AE;
   // GBK_TO_UNICODE[15269] := 16#7231;
   // GBK_TO_UNICODE[15270] := 16#B0AF;
   // GBK_TO_UNICODE[15271] := 16#9698;
   // GBK_TO_UNICODE[15272] := 16#B0B0;
   // GBK_TO_UNICODE[15273] := 16#978D;
   // GBK_TO_UNICODE[15274] := 16#B0B1;
   // GBK_TO_UNICODE[15275] := 16#6C28;
   // GBK_TO_UNICODE[15276] := 16#B0B2;
   // GBK_TO_UNICODE[15277] := 16#5B89;
   // GBK_TO_UNICODE[15278] := 16#B0B3;
   // GBK_TO_UNICODE[15279] := 16#4FFA;
   // GBK_TO_UNICODE[15280] := 16#B0B4;
   // GBK_TO_UNICODE[15281] := 16#6309;
   // GBK_TO_UNICODE[15282] := 16#B0B5;
   // GBK_TO_UNICODE[15283] := 16#6697;
   // GBK_TO_UNICODE[15284] := 16#B0B6;
   // GBK_TO_UNICODE[15285] := 16#5CB8;
   // GBK_TO_UNICODE[15286] := 16#B0B7;
   // GBK_TO_UNICODE[15287] := 16#80FA;
   // GBK_TO_UNICODE[15288] := 16#B0B8;
   // GBK_TO_UNICODE[15289] := 16#6848;
   // GBK_TO_UNICODE[15290] := 16#B0B9;
   // GBK_TO_UNICODE[15291] := 16#80AE;
   // GBK_TO_UNICODE[15292] := 16#B0BA;
   // GBK_TO_UNICODE[15293] := 16#6602;
   // GBK_TO_UNICODE[15294] := 16#B0BB;
   // GBK_TO_UNICODE[15295] := 16#76CE;
   // GBK_TO_UNICODE[15296] := 16#B0BC;
   // GBK_TO_UNICODE[15297] := 16#51F9;
   // GBK_TO_UNICODE[15298] := 16#B0BD;
   // GBK_TO_UNICODE[15299] := 16#6556;
   // GBK_TO_UNICODE[15300] := 16#B0BE;
   // GBK_TO_UNICODE[15301] := 16#71AC;
   // GBK_TO_UNICODE[15302] := 16#B0BF;
   // GBK_TO_UNICODE[15303] := 16#7FF1;
   // GBK_TO_UNICODE[15304] := 16#B0C0;
   // GBK_TO_UNICODE[15305] := 16#8884;
   // GBK_TO_UNICODE[15306] := 16#B0C1;
   // GBK_TO_UNICODE[15307] := 16#50B2;
   // GBK_TO_UNICODE[15308] := 16#B0C2;
   // GBK_TO_UNICODE[15309] := 16#5965;
   // GBK_TO_UNICODE[15310] := 16#B0C3;
   // GBK_TO_UNICODE[15311] := 16#61CA;
   // GBK_TO_UNICODE[15312] := 16#B0C4;
   // GBK_TO_UNICODE[15313] := 16#6FB3;
   // GBK_TO_UNICODE[15314] := 16#B0C5;
   // GBK_TO_UNICODE[15315] := 16#82AD;
   // GBK_TO_UNICODE[15316] := 16#B0C6;
   // GBK_TO_UNICODE[15317] := 16#634C;
   // GBK_TO_UNICODE[15318] := 16#B0C7;
   // GBK_TO_UNICODE[15319] := 16#6252;
   // GBK_TO_UNICODE[15320] := 16#B0C8;
   // GBK_TO_UNICODE[15321] := 16#53ED;
   // GBK_TO_UNICODE[15322] := 16#B0C9;
   // GBK_TO_UNICODE[15323] := 16#5427;
   // GBK_TO_UNICODE[15324] := 16#B0CA;
   // GBK_TO_UNICODE[15325] := 16#7B06;
   // GBK_TO_UNICODE[15326] := 16#B0CB;
   // GBK_TO_UNICODE[15327] := 16#516B;
   // GBK_TO_UNICODE[15328] := 16#B0CC;
   // GBK_TO_UNICODE[15329] := 16#75A4;
   // GBK_TO_UNICODE[15330] := 16#B0CD;
   // GBK_TO_UNICODE[15331] := 16#5DF4;
   // GBK_TO_UNICODE[15332] := 16#B0CE;
   // GBK_TO_UNICODE[15333] := 16#62D4;
   // GBK_TO_UNICODE[15334] := 16#B0CF;
   // GBK_TO_UNICODE[15335] := 16#8DCB;
   // GBK_TO_UNICODE[15336] := 16#B0D0;
   // GBK_TO_UNICODE[15337] := 16#9776;
   // GBK_TO_UNICODE[15338] := 16#B0D1;
   // GBK_TO_UNICODE[15339] := 16#628A;
   // GBK_TO_UNICODE[15340] := 16#B0D2;
   // GBK_TO_UNICODE[15341] := 16#8019;
   // GBK_TO_UNICODE[15342] := 16#B0D3;
   // GBK_TO_UNICODE[15343] := 16#575D;
   // GBK_TO_UNICODE[15344] := 16#B0D4;
   // GBK_TO_UNICODE[15345] := 16#9738;
   // GBK_TO_UNICODE[15346] := 16#B0D5;
   // GBK_TO_UNICODE[15347] := 16#7F62;
   // GBK_TO_UNICODE[15348] := 16#B0D6;
   // GBK_TO_UNICODE[15349] := 16#7238;
   // GBK_TO_UNICODE[15350] := 16#B0D7;
   // GBK_TO_UNICODE[15351] := 16#767D;
   // GBK_TO_UNICODE[15352] := 16#B0D8;
   // GBK_TO_UNICODE[15353] := 16#67CF;
   // GBK_TO_UNICODE[15354] := 16#B0D9;
   // GBK_TO_UNICODE[15355] := 16#767E;
   // GBK_TO_UNICODE[15356] := 16#B0DA;
   // GBK_TO_UNICODE[15357] := 16#6446;
   // GBK_TO_UNICODE[15358] := 16#B0DB;
   // GBK_TO_UNICODE[15359] := 16#4F70;
   // GBK_TO_UNICODE[15360] := 16#B0DC;
   // GBK_TO_UNICODE[15361] := 16#8D25;
   // GBK_TO_UNICODE[15362] := 16#B0DD;
   // GBK_TO_UNICODE[15363] := 16#62DC;
   // GBK_TO_UNICODE[15364] := 16#B0DE;
   // GBK_TO_UNICODE[15365] := 16#7A17;
   // GBK_TO_UNICODE[15366] := 16#B0DF;
   // GBK_TO_UNICODE[15367] := 16#6591;
   // GBK_TO_UNICODE[15368] := 16#B0E0;
   // GBK_TO_UNICODE[15369] := 16#73ED;
   // GBK_TO_UNICODE[15370] := 16#B0E1;
   // GBK_TO_UNICODE[15371] := 16#642C;
   // GBK_TO_UNICODE[15372] := 16#B0E2;
   // GBK_TO_UNICODE[15373] := 16#6273;
   // GBK_TO_UNICODE[15374] := 16#B0E3;
   // GBK_TO_UNICODE[15375] := 16#822C;
   // GBK_TO_UNICODE[15376] := 16#B0E4;
   // GBK_TO_UNICODE[15377] := 16#9881;
   // GBK_TO_UNICODE[15378] := 16#B0E5;
   // GBK_TO_UNICODE[15379] := 16#677F;
   // GBK_TO_UNICODE[15380] := 16#B0E6;
   // GBK_TO_UNICODE[15381] := 16#7248;
   // GBK_TO_UNICODE[15382] := 16#B0E7;
   // GBK_TO_UNICODE[15383] := 16#626E;
   // GBK_TO_UNICODE[15384] := 16#B0E8;
   // GBK_TO_UNICODE[15385] := 16#62CC;
   // GBK_TO_UNICODE[15386] := 16#B0E9;
   // GBK_TO_UNICODE[15387] := 16#4F34;
   // GBK_TO_UNICODE[15388] := 16#B0EA;
   // GBK_TO_UNICODE[15389] := 16#74E3;
   // GBK_TO_UNICODE[15390] := 16#B0EB;
   // GBK_TO_UNICODE[15391] := 16#534A;
   // GBK_TO_UNICODE[15392] := 16#B0EC;
   // GBK_TO_UNICODE[15393] := 16#529E;
   // GBK_TO_UNICODE[15394] := 16#B0ED;
   // GBK_TO_UNICODE[15395] := 16#7ECA;
   // GBK_TO_UNICODE[15396] := 16#B0EE;
   // GBK_TO_UNICODE[15397] := 16#90A6;
   // GBK_TO_UNICODE[15398] := 16#B0EF;
   // GBK_TO_UNICODE[15399] := 16#5E2E;
   // GBK_TO_UNICODE[15400] := 16#B0F0;
   // GBK_TO_UNICODE[15401] := 16#6886;
   // GBK_TO_UNICODE[15402] := 16#B0F1;
   // GBK_TO_UNICODE[15403] := 16#699C;
   // GBK_TO_UNICODE[15404] := 16#B0F2;
   // GBK_TO_UNICODE[15405] := 16#8180;
   // GBK_TO_UNICODE[15406] := 16#B0F3;
   // GBK_TO_UNICODE[15407] := 16#7ED1;
   // GBK_TO_UNICODE[15408] := 16#B0F4;
   // GBK_TO_UNICODE[15409] := 16#68D2;
   // GBK_TO_UNICODE[15410] := 16#B0F5;
   // GBK_TO_UNICODE[15411] := 16#78C5;
   // GBK_TO_UNICODE[15412] := 16#B0F6;
   // GBK_TO_UNICODE[15413] := 16#868C;
   // GBK_TO_UNICODE[15414] := 16#B0F7;
   // GBK_TO_UNICODE[15415] := 16#9551;
   // GBK_TO_UNICODE[15416] := 16#B0F8;
   // GBK_TO_UNICODE[15417] := 16#508D;
   // GBK_TO_UNICODE[15418] := 16#B0F9;
   // GBK_TO_UNICODE[15419] := 16#8C24;
   // GBK_TO_UNICODE[15420] := 16#B0FA;
   // GBK_TO_UNICODE[15421] := 16#82DE;
   // GBK_TO_UNICODE[15422] := 16#B0FB;
   // GBK_TO_UNICODE[15423] := 16#80DE;
   // GBK_TO_UNICODE[15424] := 16#B0FC;
   // GBK_TO_UNICODE[15425] := 16#5305;
   // GBK_TO_UNICODE[15426] := 16#B0FD;
   // GBK_TO_UNICODE[15427] := 16#8912;
   // GBK_TO_UNICODE[15428] := 16#B0FE;
   // GBK_TO_UNICODE[15429] := 16#5265;
   // GBK_TO_UNICODE[15430] := 16#B140;
   // GBK_TO_UNICODE[15431] := 16#76C4;
   // GBK_TO_UNICODE[15432] := 16#B141;
   // GBK_TO_UNICODE[15433] := 16#76C7;
   // GBK_TO_UNICODE[15434] := 16#B142;
   // GBK_TO_UNICODE[15435] := 16#76C9;
   // GBK_TO_UNICODE[15436] := 16#B143;
   // GBK_TO_UNICODE[15437] := 16#76CB;
   // GBK_TO_UNICODE[15438] := 16#B144;
   // GBK_TO_UNICODE[15439] := 16#76CC;
   // GBK_TO_UNICODE[15440] := 16#B145;
   // GBK_TO_UNICODE[15441] := 16#76D3;
   // GBK_TO_UNICODE[15442] := 16#B146;
   // GBK_TO_UNICODE[15443] := 16#76D5;
   // GBK_TO_UNICODE[15444] := 16#B147;
   // GBK_TO_UNICODE[15445] := 16#76D9;
   // GBK_TO_UNICODE[15446] := 16#B148;
   // GBK_TO_UNICODE[15447] := 16#76DA;
   // GBK_TO_UNICODE[15448] := 16#B149;
   // GBK_TO_UNICODE[15449] := 16#76DC;
   // GBK_TO_UNICODE[15450] := 16#B14A;
   // GBK_TO_UNICODE[15451] := 16#76DD;
   // GBK_TO_UNICODE[15452] := 16#B14B;
   // GBK_TO_UNICODE[15453] := 16#76DE;
   // GBK_TO_UNICODE[15454] := 16#B14C;
   // GBK_TO_UNICODE[15455] := 16#76E0;
   // GBK_TO_UNICODE[15456] := 16#B14D;
   // GBK_TO_UNICODE[15457] := 16#76E1;
   // GBK_TO_UNICODE[15458] := 16#B14E;
   // GBK_TO_UNICODE[15459] := 16#76E2;
   // GBK_TO_UNICODE[15460] := 16#B14F;
   // GBK_TO_UNICODE[15461] := 16#76E3;
   // GBK_TO_UNICODE[15462] := 16#B150;
   // GBK_TO_UNICODE[15463] := 16#76E4;
   // GBK_TO_UNICODE[15464] := 16#B151;
   // GBK_TO_UNICODE[15465] := 16#76E6;
   // GBK_TO_UNICODE[15466] := 16#B152;
   // GBK_TO_UNICODE[15467] := 16#76E7;
   // GBK_TO_UNICODE[15468] := 16#B153;
   // GBK_TO_UNICODE[15469] := 16#76E8;
   // GBK_TO_UNICODE[15470] := 16#B154;
   // GBK_TO_UNICODE[15471] := 16#76E9;
   // GBK_TO_UNICODE[15472] := 16#B155;
   // GBK_TO_UNICODE[15473] := 16#76EA;
   // GBK_TO_UNICODE[15474] := 16#B156;
   // GBK_TO_UNICODE[15475] := 16#76EB;
   // GBK_TO_UNICODE[15476] := 16#B157;
   // GBK_TO_UNICODE[15477] := 16#76EC;
   // GBK_TO_UNICODE[15478] := 16#B158;
   // GBK_TO_UNICODE[15479] := 16#76ED;
   // GBK_TO_UNICODE[15480] := 16#B159;
   // GBK_TO_UNICODE[15481] := 16#76F0;
   // GBK_TO_UNICODE[15482] := 16#B15A;
   // GBK_TO_UNICODE[15483] := 16#76F3;
   // GBK_TO_UNICODE[15484] := 16#B15B;
   // GBK_TO_UNICODE[15485] := 16#76F5;
   // GBK_TO_UNICODE[15486] := 16#B15C;
   // GBK_TO_UNICODE[15487] := 16#76F6;
   // GBK_TO_UNICODE[15488] := 16#B15D;
   // GBK_TO_UNICODE[15489] := 16#76F7;
   // GBK_TO_UNICODE[15490] := 16#B15E;
   // GBK_TO_UNICODE[15491] := 16#76FA;
   // GBK_TO_UNICODE[15492] := 16#B15F;
   // GBK_TO_UNICODE[15493] := 16#76FB;
   // GBK_TO_UNICODE[15494] := 16#B160;
   // GBK_TO_UNICODE[15495] := 16#76FD;
   // GBK_TO_UNICODE[15496] := 16#B161;
   // GBK_TO_UNICODE[15497] := 16#76FF;
   // GBK_TO_UNICODE[15498] := 16#B162;
   // GBK_TO_UNICODE[15499] := 16#7700;
   // GBK_TO_UNICODE[15500] := 16#B163;
   // GBK_TO_UNICODE[15501] := 16#7702;
   // GBK_TO_UNICODE[15502] := 16#B164;
   // GBK_TO_UNICODE[15503] := 16#7703;
   // GBK_TO_UNICODE[15504] := 16#B165;
   // GBK_TO_UNICODE[15505] := 16#7705;
   // GBK_TO_UNICODE[15506] := 16#B166;
   // GBK_TO_UNICODE[15507] := 16#7706;
   // GBK_TO_UNICODE[15508] := 16#B167;
   // GBK_TO_UNICODE[15509] := 16#770A;
   // GBK_TO_UNICODE[15510] := 16#B168;
   // GBK_TO_UNICODE[15511] := 16#770C;
   // GBK_TO_UNICODE[15512] := 16#B169;
   // GBK_TO_UNICODE[15513] := 16#770E;
   // GBK_TO_UNICODE[15514] := 16#B16A;
   // GBK_TO_UNICODE[15515] := 16#770F;
   // GBK_TO_UNICODE[15516] := 16#B16B;
   // GBK_TO_UNICODE[15517] := 16#7710;
   // GBK_TO_UNICODE[15518] := 16#B16C;
   // GBK_TO_UNICODE[15519] := 16#7711;
   // GBK_TO_UNICODE[15520] := 16#B16D;
   // GBK_TO_UNICODE[15521] := 16#7712;
   // GBK_TO_UNICODE[15522] := 16#B16E;
   // GBK_TO_UNICODE[15523] := 16#7713;
   // GBK_TO_UNICODE[15524] := 16#B16F;
   // GBK_TO_UNICODE[15525] := 16#7714;
   // GBK_TO_UNICODE[15526] := 16#B170;
   // GBK_TO_UNICODE[15527] := 16#7715;
   // GBK_TO_UNICODE[15528] := 16#B171;
   // GBK_TO_UNICODE[15529] := 16#7716;
   // GBK_TO_UNICODE[15530] := 16#B172;
   // GBK_TO_UNICODE[15531] := 16#7717;
   // GBK_TO_UNICODE[15532] := 16#B173;
   // GBK_TO_UNICODE[15533] := 16#7718;
   // GBK_TO_UNICODE[15534] := 16#B174;
   // GBK_TO_UNICODE[15535] := 16#771B;
   // GBK_TO_UNICODE[15536] := 16#B175;
   // GBK_TO_UNICODE[15537] := 16#771C;
   // GBK_TO_UNICODE[15538] := 16#B176;
   // GBK_TO_UNICODE[15539] := 16#771D;
   // GBK_TO_UNICODE[15540] := 16#B177;
   // GBK_TO_UNICODE[15541] := 16#771E;
   // GBK_TO_UNICODE[15542] := 16#B178;
   // GBK_TO_UNICODE[15543] := 16#7721;
   // GBK_TO_UNICODE[15544] := 16#B179;
   // GBK_TO_UNICODE[15545] := 16#7723;
   // GBK_TO_UNICODE[15546] := 16#B17A;
   // GBK_TO_UNICODE[15547] := 16#7724;
   // GBK_TO_UNICODE[15548] := 16#B17B;
   // GBK_TO_UNICODE[15549] := 16#7725;
   // GBK_TO_UNICODE[15550] := 16#B17C;
   // GBK_TO_UNICODE[15551] := 16#7727;
   // GBK_TO_UNICODE[15552] := 16#B17D;
   // GBK_TO_UNICODE[15553] := 16#772A;
   // GBK_TO_UNICODE[15554] := 16#B17E;
   // GBK_TO_UNICODE[15555] := 16#772B;
   // GBK_TO_UNICODE[15556] := 16#B180;
   // GBK_TO_UNICODE[15557] := 16#772C;
   // GBK_TO_UNICODE[15558] := 16#B181;
   // GBK_TO_UNICODE[15559] := 16#772E;
   // GBK_TO_UNICODE[15560] := 16#B182;
   // GBK_TO_UNICODE[15561] := 16#7730;
   // GBK_TO_UNICODE[15562] := 16#B183;
   // GBK_TO_UNICODE[15563] := 16#7731;
   // GBK_TO_UNICODE[15564] := 16#B184;
   // GBK_TO_UNICODE[15565] := 16#7732;
   // GBK_TO_UNICODE[15566] := 16#B185;
   // GBK_TO_UNICODE[15567] := 16#7733;
   // GBK_TO_UNICODE[15568] := 16#B186;
   // GBK_TO_UNICODE[15569] := 16#7734;
   // GBK_TO_UNICODE[15570] := 16#B187;
   // GBK_TO_UNICODE[15571] := 16#7739;
   // GBK_TO_UNICODE[15572] := 16#B188;
   // GBK_TO_UNICODE[15573] := 16#773B;
   // GBK_TO_UNICODE[15574] := 16#B189;
   // GBK_TO_UNICODE[15575] := 16#773D;
   // GBK_TO_UNICODE[15576] := 16#B18A;
   // GBK_TO_UNICODE[15577] := 16#773E;
   // GBK_TO_UNICODE[15578] := 16#B18B;
   // GBK_TO_UNICODE[15579] := 16#773F;
   // GBK_TO_UNICODE[15580] := 16#B18C;
   // GBK_TO_UNICODE[15581] := 16#7742;
   // GBK_TO_UNICODE[15582] := 16#B18D;
   // GBK_TO_UNICODE[15583] := 16#7744;
   // GBK_TO_UNICODE[15584] := 16#B18E;
   // GBK_TO_UNICODE[15585] := 16#7745;
   // GBK_TO_UNICODE[15586] := 16#B18F;
   // GBK_TO_UNICODE[15587] := 16#7746;
   // GBK_TO_UNICODE[15588] := 16#B190;
   // GBK_TO_UNICODE[15589] := 16#7748;
   // GBK_TO_UNICODE[15590] := 16#B191;
   // GBK_TO_UNICODE[15591] := 16#7749;
   // GBK_TO_UNICODE[15592] := 16#B192;
   // GBK_TO_UNICODE[15593] := 16#774A;
   // GBK_TO_UNICODE[15594] := 16#B193;
   // GBK_TO_UNICODE[15595] := 16#774B;
   // GBK_TO_UNICODE[15596] := 16#B194;
   // GBK_TO_UNICODE[15597] := 16#774C;
   // GBK_TO_UNICODE[15598] := 16#B195;
   // GBK_TO_UNICODE[15599] := 16#774D;
   // GBK_TO_UNICODE[15600] := 16#B196;
   // GBK_TO_UNICODE[15601] := 16#774E;
   // GBK_TO_UNICODE[15602] := 16#B197;
   // GBK_TO_UNICODE[15603] := 16#774F;
   // GBK_TO_UNICODE[15604] := 16#B198;
   // GBK_TO_UNICODE[15605] := 16#7752;
   // GBK_TO_UNICODE[15606] := 16#B199;
   // GBK_TO_UNICODE[15607] := 16#7753;
   // GBK_TO_UNICODE[15608] := 16#B19A;
   // GBK_TO_UNICODE[15609] := 16#7754;
   // GBK_TO_UNICODE[15610] := 16#B19B;
   // GBK_TO_UNICODE[15611] := 16#7755;
   // GBK_TO_UNICODE[15612] := 16#B19C;
   // GBK_TO_UNICODE[15613] := 16#7756;
   // GBK_TO_UNICODE[15614] := 16#B19D;
   // GBK_TO_UNICODE[15615] := 16#7757;
   // GBK_TO_UNICODE[15616] := 16#B19E;
   // GBK_TO_UNICODE[15617] := 16#7758;
   // GBK_TO_UNICODE[15618] := 16#B19F;
   // GBK_TO_UNICODE[15619] := 16#7759;
   // GBK_TO_UNICODE[15620] := 16#B1A0;
   // GBK_TO_UNICODE[15621] := 16#775C;
   // GBK_TO_UNICODE[15622] := 16#B1A1;
   // GBK_TO_UNICODE[15623] := 16#8584;
   // GBK_TO_UNICODE[15624] := 16#B1A2;
   // GBK_TO_UNICODE[15625] := 16#96F9;
   // GBK_TO_UNICODE[15626] := 16#B1A3;
   // GBK_TO_UNICODE[15627] := 16#4FDD;
   // GBK_TO_UNICODE[15628] := 16#B1A4;
   // GBK_TO_UNICODE[15629] := 16#5821;
   // GBK_TO_UNICODE[15630] := 16#B1A5;
   // GBK_TO_UNICODE[15631] := 16#9971;
   // GBK_TO_UNICODE[15632] := 16#B1A6;
   // GBK_TO_UNICODE[15633] := 16#5B9D;
   // GBK_TO_UNICODE[15634] := 16#B1A7;
   // GBK_TO_UNICODE[15635] := 16#62B1;
   // GBK_TO_UNICODE[15636] := 16#B1A8;
   // GBK_TO_UNICODE[15637] := 16#62A5;
   // GBK_TO_UNICODE[15638] := 16#B1A9;
   // GBK_TO_UNICODE[15639] := 16#66B4;
   // GBK_TO_UNICODE[15640] := 16#B1AA;
   // GBK_TO_UNICODE[15641] := 16#8C79;
   // GBK_TO_UNICODE[15642] := 16#B1AB;
   // GBK_TO_UNICODE[15643] := 16#9C8D;
   // GBK_TO_UNICODE[15644] := 16#B1AC;
   // GBK_TO_UNICODE[15645] := 16#7206;
   // GBK_TO_UNICODE[15646] := 16#B1AD;
   // GBK_TO_UNICODE[15647] := 16#676F;
   // GBK_TO_UNICODE[15648] := 16#B1AE;
   // GBK_TO_UNICODE[15649] := 16#7891;
   // GBK_TO_UNICODE[15650] := 16#B1AF;
   // GBK_TO_UNICODE[15651] := 16#60B2;
   // GBK_TO_UNICODE[15652] := 16#B1B0;
   // GBK_TO_UNICODE[15653] := 16#5351;
   // GBK_TO_UNICODE[15654] := 16#B1B1;
   // GBK_TO_UNICODE[15655] := 16#5317;
   // GBK_TO_UNICODE[15656] := 16#B1B2;
   // GBK_TO_UNICODE[15657] := 16#8F88;
   // GBK_TO_UNICODE[15658] := 16#B1B3;
   // GBK_TO_UNICODE[15659] := 16#80CC;
   // GBK_TO_UNICODE[15660] := 16#B1B4;
   // GBK_TO_UNICODE[15661] := 16#8D1D;
   // GBK_TO_UNICODE[15662] := 16#B1B5;
   // GBK_TO_UNICODE[15663] := 16#94A1;
   // GBK_TO_UNICODE[15664] := 16#B1B6;
   // GBK_TO_UNICODE[15665] := 16#500D;
   // GBK_TO_UNICODE[15666] := 16#B1B7;
   // GBK_TO_UNICODE[15667] := 16#72C8;
   // GBK_TO_UNICODE[15668] := 16#B1B8;
   // GBK_TO_UNICODE[15669] := 16#5907;
   // GBK_TO_UNICODE[15670] := 16#B1B9;
   // GBK_TO_UNICODE[15671] := 16#60EB;
   // GBK_TO_UNICODE[15672] := 16#B1BA;
   // GBK_TO_UNICODE[15673] := 16#7119;
   // GBK_TO_UNICODE[15674] := 16#B1BB;
   // GBK_TO_UNICODE[15675] := 16#88AB;
   // GBK_TO_UNICODE[15676] := 16#B1BC;
   // GBK_TO_UNICODE[15677] := 16#5954;
   // GBK_TO_UNICODE[15678] := 16#B1BD;
   // GBK_TO_UNICODE[15679] := 16#82EF;
   // GBK_TO_UNICODE[15680] := 16#B1BE;
   // GBK_TO_UNICODE[15681] := 16#672C;
   // GBK_TO_UNICODE[15682] := 16#B1BF;
   // GBK_TO_UNICODE[15683] := 16#7B28;
   // GBK_TO_UNICODE[15684] := 16#B1C0;
   // GBK_TO_UNICODE[15685] := 16#5D29;
   // GBK_TO_UNICODE[15686] := 16#B1C1;
   // GBK_TO_UNICODE[15687] := 16#7EF7;
   // GBK_TO_UNICODE[15688] := 16#B1C2;
   // GBK_TO_UNICODE[15689] := 16#752D;
   // GBK_TO_UNICODE[15690] := 16#B1C3;
   // GBK_TO_UNICODE[15691] := 16#6CF5;
   // GBK_TO_UNICODE[15692] := 16#B1C4;
   // GBK_TO_UNICODE[15693] := 16#8E66;
   // GBK_TO_UNICODE[15694] := 16#B1C5;
   // GBK_TO_UNICODE[15695] := 16#8FF8;
   // GBK_TO_UNICODE[15696] := 16#B1C6;
   // GBK_TO_UNICODE[15697] := 16#903C;
   // GBK_TO_UNICODE[15698] := 16#B1C7;
   // GBK_TO_UNICODE[15699] := 16#9F3B;
   // GBK_TO_UNICODE[15700] := 16#B1C8;
   // GBK_TO_UNICODE[15701] := 16#6BD4;
   // GBK_TO_UNICODE[15702] := 16#B1C9;
   // GBK_TO_UNICODE[15703] := 16#9119;
   // GBK_TO_UNICODE[15704] := 16#B1CA;
   // GBK_TO_UNICODE[15705] := 16#7B14;
   // GBK_TO_UNICODE[15706] := 16#B1CB;
   // GBK_TO_UNICODE[15707] := 16#5F7C;
   // GBK_TO_UNICODE[15708] := 16#B1CC;
   // GBK_TO_UNICODE[15709] := 16#78A7;
   // GBK_TO_UNICODE[15710] := 16#B1CD;
   // GBK_TO_UNICODE[15711] := 16#84D6;
   // GBK_TO_UNICODE[15712] := 16#B1CE;
   // GBK_TO_UNICODE[15713] := 16#853D;
   // GBK_TO_UNICODE[15714] := 16#B1CF;
   // GBK_TO_UNICODE[15715] := 16#6BD5;
   // GBK_TO_UNICODE[15716] := 16#B1D0;
   // GBK_TO_UNICODE[15717] := 16#6BD9;
   // GBK_TO_UNICODE[15718] := 16#B1D1;
   // GBK_TO_UNICODE[15719] := 16#6BD6;
   // GBK_TO_UNICODE[15720] := 16#B1D2;
   // GBK_TO_UNICODE[15721] := 16#5E01;
   // GBK_TO_UNICODE[15722] := 16#B1D3;
   // GBK_TO_UNICODE[15723] := 16#5E87;
   // GBK_TO_UNICODE[15724] := 16#B1D4;
   // GBK_TO_UNICODE[15725] := 16#75F9;
   // GBK_TO_UNICODE[15726] := 16#B1D5;
   // GBK_TO_UNICODE[15727] := 16#95ED;
   // GBK_TO_UNICODE[15728] := 16#B1D6;
   // GBK_TO_UNICODE[15729] := 16#655D;
   // GBK_TO_UNICODE[15730] := 16#B1D7;
   // GBK_TO_UNICODE[15731] := 16#5F0A;
   // GBK_TO_UNICODE[15732] := 16#B1D8;
   // GBK_TO_UNICODE[15733] := 16#5FC5;
   // GBK_TO_UNICODE[15734] := 16#B1D9;
   // GBK_TO_UNICODE[15735] := 16#8F9F;
   // GBK_TO_UNICODE[15736] := 16#B1DA;
   // GBK_TO_UNICODE[15737] := 16#58C1;
   // GBK_TO_UNICODE[15738] := 16#B1DB;
   // GBK_TO_UNICODE[15739] := 16#81C2;
   // GBK_TO_UNICODE[15740] := 16#B1DC;
   // GBK_TO_UNICODE[15741] := 16#907F;
   // GBK_TO_UNICODE[15742] := 16#B1DD;
   // GBK_TO_UNICODE[15743] := 16#965B;
   // GBK_TO_UNICODE[15744] := 16#B1DE;
   // GBK_TO_UNICODE[15745] := 16#97AD;
   // GBK_TO_UNICODE[15746] := 16#B1DF;
   // GBK_TO_UNICODE[15747] := 16#8FB9;
   // GBK_TO_UNICODE[15748] := 16#B1E0;
   // GBK_TO_UNICODE[15749] := 16#7F16;
   // GBK_TO_UNICODE[15750] := 16#B1E1;
   // GBK_TO_UNICODE[15751] := 16#8D2C;
   // GBK_TO_UNICODE[15752] := 16#B1E2;
   // GBK_TO_UNICODE[15753] := 16#6241;
   // GBK_TO_UNICODE[15754] := 16#B1E3;
   // GBK_TO_UNICODE[15755] := 16#4FBF;
   // GBK_TO_UNICODE[15756] := 16#B1E4;
   // GBK_TO_UNICODE[15757] := 16#53D8;
   // GBK_TO_UNICODE[15758] := 16#B1E5;
   // GBK_TO_UNICODE[15759] := 16#535E;
   // GBK_TO_UNICODE[15760] := 16#B1E6;
   // GBK_TO_UNICODE[15761] := 16#8FA8;
   // GBK_TO_UNICODE[15762] := 16#B1E7;
   // GBK_TO_UNICODE[15763] := 16#8FA9;
   // GBK_TO_UNICODE[15764] := 16#B1E8;
   // GBK_TO_UNICODE[15765] := 16#8FAB;
   // GBK_TO_UNICODE[15766] := 16#B1E9;
   // GBK_TO_UNICODE[15767] := 16#904D;
   // GBK_TO_UNICODE[15768] := 16#B1EA;
   // GBK_TO_UNICODE[15769] := 16#6807;
   // GBK_TO_UNICODE[15770] := 16#B1EB;
   // GBK_TO_UNICODE[15771] := 16#5F6A;
   // GBK_TO_UNICODE[15772] := 16#B1EC;
   // GBK_TO_UNICODE[15773] := 16#8198;
   // GBK_TO_UNICODE[15774] := 16#B1ED;
   // GBK_TO_UNICODE[15775] := 16#8868;
   // GBK_TO_UNICODE[15776] := 16#B1EE;
   // GBK_TO_UNICODE[15777] := 16#9CD6;
   // GBK_TO_UNICODE[15778] := 16#B1EF;
   // GBK_TO_UNICODE[15779] := 16#618B;
   // GBK_TO_UNICODE[15780] := 16#B1F0;
   // GBK_TO_UNICODE[15781] := 16#522B;
   // GBK_TO_UNICODE[15782] := 16#B1F1;
   // GBK_TO_UNICODE[15783] := 16#762A;
   // GBK_TO_UNICODE[15784] := 16#B1F2;
   // GBK_TO_UNICODE[15785] := 16#5F6C;
   // GBK_TO_UNICODE[15786] := 16#B1F3;
   // GBK_TO_UNICODE[15787] := 16#658C;
   // GBK_TO_UNICODE[15788] := 16#B1F4;
   // GBK_TO_UNICODE[15789] := 16#6FD2;
   // GBK_TO_UNICODE[15790] := 16#B1F5;
   // GBK_TO_UNICODE[15791] := 16#6EE8;
   // GBK_TO_UNICODE[15792] := 16#B1F6;
   // GBK_TO_UNICODE[15793] := 16#5BBE;
   // GBK_TO_UNICODE[15794] := 16#B1F7;
   // GBK_TO_UNICODE[15795] := 16#6448;
   // GBK_TO_UNICODE[15796] := 16#B1F8;
   // GBK_TO_UNICODE[15797] := 16#5175;
   // GBK_TO_UNICODE[15798] := 16#B1F9;
   // GBK_TO_UNICODE[15799] := 16#51B0;
   // GBK_TO_UNICODE[15800] := 16#B1FA;
   // GBK_TO_UNICODE[15801] := 16#67C4;
   // GBK_TO_UNICODE[15802] := 16#B1FB;
   // GBK_TO_UNICODE[15803] := 16#4E19;
   // GBK_TO_UNICODE[15804] := 16#B1FC;
   // GBK_TO_UNICODE[15805] := 16#79C9;
   // GBK_TO_UNICODE[15806] := 16#B1FD;
   // GBK_TO_UNICODE[15807] := 16#997C;
   // GBK_TO_UNICODE[15808] := 16#B1FE;
   // GBK_TO_UNICODE[15809] := 16#70B3;
   // GBK_TO_UNICODE[15810] := 16#B240;
   // GBK_TO_UNICODE[15811] := 16#775D;
   // GBK_TO_UNICODE[15812] := 16#B241;
   // GBK_TO_UNICODE[15813] := 16#775E;
   // GBK_TO_UNICODE[15814] := 16#B242;
   // GBK_TO_UNICODE[15815] := 16#775F;
   // GBK_TO_UNICODE[15816] := 16#B243;
   // GBK_TO_UNICODE[15817] := 16#7760;
   // GBK_TO_UNICODE[15818] := 16#B244;
   // GBK_TO_UNICODE[15819] := 16#7764;
   // GBK_TO_UNICODE[15820] := 16#B245;
   // GBK_TO_UNICODE[15821] := 16#7767;
   // GBK_TO_UNICODE[15822] := 16#B246;
   // GBK_TO_UNICODE[15823] := 16#7769;
   // GBK_TO_UNICODE[15824] := 16#B247;
   // GBK_TO_UNICODE[15825] := 16#776A;
   // GBK_TO_UNICODE[15826] := 16#B248;
   // GBK_TO_UNICODE[15827] := 16#776D;
   // GBK_TO_UNICODE[15828] := 16#B249;
   // GBK_TO_UNICODE[15829] := 16#776E;
   // GBK_TO_UNICODE[15830] := 16#B24A;
   // GBK_TO_UNICODE[15831] := 16#776F;
   // GBK_TO_UNICODE[15832] := 16#B24B;
   // GBK_TO_UNICODE[15833] := 16#7770;
   // GBK_TO_UNICODE[15834] := 16#B24C;
   // GBK_TO_UNICODE[15835] := 16#7771;
   // GBK_TO_UNICODE[15836] := 16#B24D;
   // GBK_TO_UNICODE[15837] := 16#7772;
   // GBK_TO_UNICODE[15838] := 16#B24E;
   // GBK_TO_UNICODE[15839] := 16#7773;
   // GBK_TO_UNICODE[15840] := 16#B24F;
   // GBK_TO_UNICODE[15841] := 16#7774;
   // GBK_TO_UNICODE[15842] := 16#B250;
   // GBK_TO_UNICODE[15843] := 16#7775;
   // GBK_TO_UNICODE[15844] := 16#B251;
   // GBK_TO_UNICODE[15845] := 16#7776;
   // GBK_TO_UNICODE[15846] := 16#B252;
   // GBK_TO_UNICODE[15847] := 16#7777;
   // GBK_TO_UNICODE[15848] := 16#B253;
   // GBK_TO_UNICODE[15849] := 16#7778;
   // GBK_TO_UNICODE[15850] := 16#B254;
   // GBK_TO_UNICODE[15851] := 16#777A;
   // GBK_TO_UNICODE[15852] := 16#B255;
   // GBK_TO_UNICODE[15853] := 16#777B;
   // GBK_TO_UNICODE[15854] := 16#B256;
   // GBK_TO_UNICODE[15855] := 16#777C;
   // GBK_TO_UNICODE[15856] := 16#B257;
   // GBK_TO_UNICODE[15857] := 16#7781;
   // GBK_TO_UNICODE[15858] := 16#B258;
   // GBK_TO_UNICODE[15859] := 16#7782;
   // GBK_TO_UNICODE[15860] := 16#B259;
   // GBK_TO_UNICODE[15861] := 16#7783;
   // GBK_TO_UNICODE[15862] := 16#B25A;
   // GBK_TO_UNICODE[15863] := 16#7786;
   // GBK_TO_UNICODE[15864] := 16#B25B;
   // GBK_TO_UNICODE[15865] := 16#7787;
   // GBK_TO_UNICODE[15866] := 16#B25C;
   // GBK_TO_UNICODE[15867] := 16#7788;
   // GBK_TO_UNICODE[15868] := 16#B25D;
   // GBK_TO_UNICODE[15869] := 16#7789;
   // GBK_TO_UNICODE[15870] := 16#B25E;
   // GBK_TO_UNICODE[15871] := 16#778A;
   // GBK_TO_UNICODE[15872] := 16#B25F;
   // GBK_TO_UNICODE[15873] := 16#778B;
   // GBK_TO_UNICODE[15874] := 16#B260;
   // GBK_TO_UNICODE[15875] := 16#778F;
   // GBK_TO_UNICODE[15876] := 16#B261;
   // GBK_TO_UNICODE[15877] := 16#7790;
   // GBK_TO_UNICODE[15878] := 16#B262;
   // GBK_TO_UNICODE[15879] := 16#7793;
   // GBK_TO_UNICODE[15880] := 16#B263;
   // GBK_TO_UNICODE[15881] := 16#7794;
   // GBK_TO_UNICODE[15882] := 16#B264;
   // GBK_TO_UNICODE[15883] := 16#7795;
   // GBK_TO_UNICODE[15884] := 16#B265;
   // GBK_TO_UNICODE[15885] := 16#7796;
   // GBK_TO_UNICODE[15886] := 16#B266;
   // GBK_TO_UNICODE[15887] := 16#7797;
   // GBK_TO_UNICODE[15888] := 16#B267;
   // GBK_TO_UNICODE[15889] := 16#7798;
   // GBK_TO_UNICODE[15890] := 16#B268;
   // GBK_TO_UNICODE[15891] := 16#7799;
   // GBK_TO_UNICODE[15892] := 16#B269;
   // GBK_TO_UNICODE[15893] := 16#779A;
   // GBK_TO_UNICODE[15894] := 16#B26A;
   // GBK_TO_UNICODE[15895] := 16#779B;
   // GBK_TO_UNICODE[15896] := 16#B26B;
   // GBK_TO_UNICODE[15897] := 16#779C;
   // GBK_TO_UNICODE[15898] := 16#B26C;
   // GBK_TO_UNICODE[15899] := 16#779D;
   // GBK_TO_UNICODE[15900] := 16#B26D;
   // GBK_TO_UNICODE[15901] := 16#779E;
   // GBK_TO_UNICODE[15902] := 16#B26E;
   // GBK_TO_UNICODE[15903] := 16#77A1;
   // GBK_TO_UNICODE[15904] := 16#B26F;
   // GBK_TO_UNICODE[15905] := 16#77A3;
   // GBK_TO_UNICODE[15906] := 16#B270;
   // GBK_TO_UNICODE[15907] := 16#77A4;
   // GBK_TO_UNICODE[15908] := 16#B271;
   // GBK_TO_UNICODE[15909] := 16#77A6;
   // GBK_TO_UNICODE[15910] := 16#B272;
   // GBK_TO_UNICODE[15911] := 16#77A8;
   // GBK_TO_UNICODE[15912] := 16#B273;
   // GBK_TO_UNICODE[15913] := 16#77AB;
   // GBK_TO_UNICODE[15914] := 16#B274;
   // GBK_TO_UNICODE[15915] := 16#77AD;
   // GBK_TO_UNICODE[15916] := 16#B275;
   // GBK_TO_UNICODE[15917] := 16#77AE;
   // GBK_TO_UNICODE[15918] := 16#B276;
   // GBK_TO_UNICODE[15919] := 16#77AF;
   // GBK_TO_UNICODE[15920] := 16#B277;
   // GBK_TO_UNICODE[15921] := 16#77B1;
   // GBK_TO_UNICODE[15922] := 16#B278;
   // GBK_TO_UNICODE[15923] := 16#77B2;
   // GBK_TO_UNICODE[15924] := 16#B279;
   // GBK_TO_UNICODE[15925] := 16#77B4;
   // GBK_TO_UNICODE[15926] := 16#B27A;
   // GBK_TO_UNICODE[15927] := 16#77B6;
   // GBK_TO_UNICODE[15928] := 16#B27B;
   // GBK_TO_UNICODE[15929] := 16#77B7;
   // GBK_TO_UNICODE[15930] := 16#B27C;
   // GBK_TO_UNICODE[15931] := 16#77B8;
   // GBK_TO_UNICODE[15932] := 16#B27D;
   // GBK_TO_UNICODE[15933] := 16#77B9;
   // GBK_TO_UNICODE[15934] := 16#B27E;
   // GBK_TO_UNICODE[15935] := 16#77BA;
   // GBK_TO_UNICODE[15936] := 16#B280;
   // GBK_TO_UNICODE[15937] := 16#77BC;
   // GBK_TO_UNICODE[15938] := 16#B281;
   // GBK_TO_UNICODE[15939] := 16#77BE;
   // GBK_TO_UNICODE[15940] := 16#B282;
   // GBK_TO_UNICODE[15941] := 16#77C0;
   // GBK_TO_UNICODE[15942] := 16#B283;
   // GBK_TO_UNICODE[15943] := 16#77C1;
   // GBK_TO_UNICODE[15944] := 16#B284;
   // GBK_TO_UNICODE[15945] := 16#77C2;
   // GBK_TO_UNICODE[15946] := 16#B285;
   // GBK_TO_UNICODE[15947] := 16#77C3;
   // GBK_TO_UNICODE[15948] := 16#B286;
   // GBK_TO_UNICODE[15949] := 16#77C4;
   // GBK_TO_UNICODE[15950] := 16#B287;
   // GBK_TO_UNICODE[15951] := 16#77C5;
   // GBK_TO_UNICODE[15952] := 16#B288;
   // GBK_TO_UNICODE[15953] := 16#77C6;
   // GBK_TO_UNICODE[15954] := 16#B289;
   // GBK_TO_UNICODE[15955] := 16#77C7;
   // GBK_TO_UNICODE[15956] := 16#B28A;
   // GBK_TO_UNICODE[15957] := 16#77C8;
   // GBK_TO_UNICODE[15958] := 16#B28B;
   // GBK_TO_UNICODE[15959] := 16#77C9;
   // GBK_TO_UNICODE[15960] := 16#B28C;
   // GBK_TO_UNICODE[15961] := 16#77CA;
   // GBK_TO_UNICODE[15962] := 16#B28D;
   // GBK_TO_UNICODE[15963] := 16#77CB;
   // GBK_TO_UNICODE[15964] := 16#B28E;
   // GBK_TO_UNICODE[15965] := 16#77CC;
   // GBK_TO_UNICODE[15966] := 16#B28F;
   // GBK_TO_UNICODE[15967] := 16#77CE;
   // GBK_TO_UNICODE[15968] := 16#B290;
   // GBK_TO_UNICODE[15969] := 16#77CF;
   // GBK_TO_UNICODE[15970] := 16#B291;
   // GBK_TO_UNICODE[15971] := 16#77D0;
   // GBK_TO_UNICODE[15972] := 16#B292;
   // GBK_TO_UNICODE[15973] := 16#77D1;
   // GBK_TO_UNICODE[15974] := 16#B293;
   // GBK_TO_UNICODE[15975] := 16#77D2;
   // GBK_TO_UNICODE[15976] := 16#B294;
   // GBK_TO_UNICODE[15977] := 16#77D3;
   // GBK_TO_UNICODE[15978] := 16#B295;
   // GBK_TO_UNICODE[15979] := 16#77D4;
   // GBK_TO_UNICODE[15980] := 16#B296;
   // GBK_TO_UNICODE[15981] := 16#77D5;
   // GBK_TO_UNICODE[15982] := 16#B297;
   // GBK_TO_UNICODE[15983] := 16#77D6;
   // GBK_TO_UNICODE[15984] := 16#B298;
   // GBK_TO_UNICODE[15985] := 16#77D8;
   // GBK_TO_UNICODE[15986] := 16#B299;
   // GBK_TO_UNICODE[15987] := 16#77D9;
   // GBK_TO_UNICODE[15988] := 16#B29A;
   // GBK_TO_UNICODE[15989] := 16#77DA;
   // GBK_TO_UNICODE[15990] := 16#B29B;
   // GBK_TO_UNICODE[15991] := 16#77DD;
   // GBK_TO_UNICODE[15992] := 16#B29C;
   // GBK_TO_UNICODE[15993] := 16#77DE;
   // GBK_TO_UNICODE[15994] := 16#B29D;
   // GBK_TO_UNICODE[15995] := 16#77DF;
   // GBK_TO_UNICODE[15996] := 16#B29E;
   // GBK_TO_UNICODE[15997] := 16#77E0;
   // GBK_TO_UNICODE[15998] := 16#B29F;
   // GBK_TO_UNICODE[15999] := 16#77E1;
   // GBK_TO_UNICODE[16000] := 16#B2A0;
   // GBK_TO_UNICODE[16001] := 16#77E4;
   // GBK_TO_UNICODE[16002] := 16#B2A1;
   // GBK_TO_UNICODE[16003] := 16#75C5;
   // GBK_TO_UNICODE[16004] := 16#B2A2;
   // GBK_TO_UNICODE[16005] := 16#5E76;
   // GBK_TO_UNICODE[16006] := 16#B2A3;
   // GBK_TO_UNICODE[16007] := 16#73BB;
   // GBK_TO_UNICODE[16008] := 16#B2A4;
   // GBK_TO_UNICODE[16009] := 16#83E0;
   // GBK_TO_UNICODE[16010] := 16#B2A5;
   // GBK_TO_UNICODE[16011] := 16#64AD;
   // GBK_TO_UNICODE[16012] := 16#B2A6;
   // GBK_TO_UNICODE[16013] := 16#62E8;
   // GBK_TO_UNICODE[16014] := 16#B2A7;
   // GBK_TO_UNICODE[16015] := 16#94B5;
   // GBK_TO_UNICODE[16016] := 16#B2A8;
   // GBK_TO_UNICODE[16017] := 16#6CE2;
   // GBK_TO_UNICODE[16018] := 16#B2A9;
   // GBK_TO_UNICODE[16019] := 16#535A;
   // GBK_TO_UNICODE[16020] := 16#B2AA;
   // GBK_TO_UNICODE[16021] := 16#52C3;
   // GBK_TO_UNICODE[16022] := 16#B2AB;
   // GBK_TO_UNICODE[16023] := 16#640F;
   // GBK_TO_UNICODE[16024] := 16#B2AC;
   // GBK_TO_UNICODE[16025] := 16#94C2;
   // GBK_TO_UNICODE[16026] := 16#B2AD;
   // GBK_TO_UNICODE[16027] := 16#7B94;
   // GBK_TO_UNICODE[16028] := 16#B2AE;
   // GBK_TO_UNICODE[16029] := 16#4F2F;
   // GBK_TO_UNICODE[16030] := 16#B2AF;
   // GBK_TO_UNICODE[16031] := 16#5E1B;
   // GBK_TO_UNICODE[16032] := 16#B2B0;
   // GBK_TO_UNICODE[16033] := 16#8236;
   // GBK_TO_UNICODE[16034] := 16#B2B1;
   // GBK_TO_UNICODE[16035] := 16#8116;
   // GBK_TO_UNICODE[16036] := 16#B2B2;
   // GBK_TO_UNICODE[16037] := 16#818A;
   // GBK_TO_UNICODE[16038] := 16#B2B3;
   // GBK_TO_UNICODE[16039] := 16#6E24;
   // GBK_TO_UNICODE[16040] := 16#B2B4;
   // GBK_TO_UNICODE[16041] := 16#6CCA;
   // GBK_TO_UNICODE[16042] := 16#B2B5;
   // GBK_TO_UNICODE[16043] := 16#9A73;
   // GBK_TO_UNICODE[16044] := 16#B2B6;
   // GBK_TO_UNICODE[16045] := 16#6355;
   // GBK_TO_UNICODE[16046] := 16#B2B7;
   // GBK_TO_UNICODE[16047] := 16#535C;
   // GBK_TO_UNICODE[16048] := 16#B2B8;
   // GBK_TO_UNICODE[16049] := 16#54FA;
   // GBK_TO_UNICODE[16050] := 16#B2B9;
   // GBK_TO_UNICODE[16051] := 16#8865;
   // GBK_TO_UNICODE[16052] := 16#B2BA;
   // GBK_TO_UNICODE[16053] := 16#57E0;
   // GBK_TO_UNICODE[16054] := 16#B2BB;
   // GBK_TO_UNICODE[16055] := 16#4E0D;
   // GBK_TO_UNICODE[16056] := 16#B2BC;
   // GBK_TO_UNICODE[16057] := 16#5E03;
   // GBK_TO_UNICODE[16058] := 16#B2BD;
   // GBK_TO_UNICODE[16059] := 16#6B65;
   // GBK_TO_UNICODE[16060] := 16#B2BE;
   // GBK_TO_UNICODE[16061] := 16#7C3F;
   // GBK_TO_UNICODE[16062] := 16#B2BF;
   // GBK_TO_UNICODE[16063] := 16#90E8;
   // GBK_TO_UNICODE[16064] := 16#B2C0;
   // GBK_TO_UNICODE[16065] := 16#6016;
   // GBK_TO_UNICODE[16066] := 16#B2C1;
   // GBK_TO_UNICODE[16067] := 16#64E6;
   // GBK_TO_UNICODE[16068] := 16#B2C2;
   // GBK_TO_UNICODE[16069] := 16#731C;
   // GBK_TO_UNICODE[16070] := 16#B2C3;
   // GBK_TO_UNICODE[16071] := 16#88C1;
   // GBK_TO_UNICODE[16072] := 16#B2C4;
   // GBK_TO_UNICODE[16073] := 16#6750;
   // GBK_TO_UNICODE[16074] := 16#B2C5;
   // GBK_TO_UNICODE[16075] := 16#624D;
   // GBK_TO_UNICODE[16076] := 16#B2C6;
   // GBK_TO_UNICODE[16077] := 16#8D22;
   // GBK_TO_UNICODE[16078] := 16#B2C7;
   // GBK_TO_UNICODE[16079] := 16#776C;
   // GBK_TO_UNICODE[16080] := 16#B2C8;
   // GBK_TO_UNICODE[16081] := 16#8E29;
   // GBK_TO_UNICODE[16082] := 16#B2C9;
   // GBK_TO_UNICODE[16083] := 16#91C7;
   // GBK_TO_UNICODE[16084] := 16#B2CA;
   // GBK_TO_UNICODE[16085] := 16#5F69;
   // GBK_TO_UNICODE[16086] := 16#B2CB;
   // GBK_TO_UNICODE[16087] := 16#83DC;
   // GBK_TO_UNICODE[16088] := 16#B2CC;
   // GBK_TO_UNICODE[16089] := 16#8521;
   // GBK_TO_UNICODE[16090] := 16#B2CD;
   // GBK_TO_UNICODE[16091] := 16#9910;
   // GBK_TO_UNICODE[16092] := 16#B2CE;
   // GBK_TO_UNICODE[16093] := 16#53C2;
   // GBK_TO_UNICODE[16094] := 16#B2CF;
   // GBK_TO_UNICODE[16095] := 16#8695;
   // GBK_TO_UNICODE[16096] := 16#B2D0;
   // GBK_TO_UNICODE[16097] := 16#6B8B;
   // GBK_TO_UNICODE[16098] := 16#B2D1;
   // GBK_TO_UNICODE[16099] := 16#60ED;
   // GBK_TO_UNICODE[16100] := 16#B2D2;
   // GBK_TO_UNICODE[16101] := 16#60E8;
   // GBK_TO_UNICODE[16102] := 16#B2D3;
   // GBK_TO_UNICODE[16103] := 16#707F;
   // GBK_TO_UNICODE[16104] := 16#B2D4;
   // GBK_TO_UNICODE[16105] := 16#82CD;
   // GBK_TO_UNICODE[16106] := 16#B2D5;
   // GBK_TO_UNICODE[16107] := 16#8231;
   // GBK_TO_UNICODE[16108] := 16#B2D6;
   // GBK_TO_UNICODE[16109] := 16#4ED3;
   // GBK_TO_UNICODE[16110] := 16#B2D7;
   // GBK_TO_UNICODE[16111] := 16#6CA7;
   // GBK_TO_UNICODE[16112] := 16#B2D8;
   // GBK_TO_UNICODE[16113] := 16#85CF;
   // GBK_TO_UNICODE[16114] := 16#B2D9;
   // GBK_TO_UNICODE[16115] := 16#64CD;
   // GBK_TO_UNICODE[16116] := 16#B2DA;
   // GBK_TO_UNICODE[16117] := 16#7CD9;
   // GBK_TO_UNICODE[16118] := 16#B2DB;
   // GBK_TO_UNICODE[16119] := 16#69FD;
   // GBK_TO_UNICODE[16120] := 16#B2DC;
   // GBK_TO_UNICODE[16121] := 16#66F9;
   // GBK_TO_UNICODE[16122] := 16#B2DD;
   // GBK_TO_UNICODE[16123] := 16#8349;
   // GBK_TO_UNICODE[16124] := 16#B2DE;
   // GBK_TO_UNICODE[16125] := 16#5395;
   // GBK_TO_UNICODE[16126] := 16#B2DF;
   // GBK_TO_UNICODE[16127] := 16#7B56;
   // GBK_TO_UNICODE[16128] := 16#B2E0;
   // GBK_TO_UNICODE[16129] := 16#4FA7;
   // GBK_TO_UNICODE[16130] := 16#B2E1;
   // GBK_TO_UNICODE[16131] := 16#518C;
   // GBK_TO_UNICODE[16132] := 16#B2E2;
   // GBK_TO_UNICODE[16133] := 16#6D4B;
   // GBK_TO_UNICODE[16134] := 16#B2E3;
   // GBK_TO_UNICODE[16135] := 16#5C42;
   // GBK_TO_UNICODE[16136] := 16#B2E4;
   // GBK_TO_UNICODE[16137] := 16#8E6D;
   // GBK_TO_UNICODE[16138] := 16#B2E5;
   // GBK_TO_UNICODE[16139] := 16#63D2;
   // GBK_TO_UNICODE[16140] := 16#B2E6;
   // GBK_TO_UNICODE[16141] := 16#53C9;
   // GBK_TO_UNICODE[16142] := 16#B2E7;
   // GBK_TO_UNICODE[16143] := 16#832C;
   // GBK_TO_UNICODE[16144] := 16#B2E8;
   // GBK_TO_UNICODE[16145] := 16#8336;
   // GBK_TO_UNICODE[16146] := 16#B2E9;
   // GBK_TO_UNICODE[16147] := 16#67E5;
   // GBK_TO_UNICODE[16148] := 16#B2EA;
   // GBK_TO_UNICODE[16149] := 16#78B4;
   // GBK_TO_UNICODE[16150] := 16#B2EB;
   // GBK_TO_UNICODE[16151] := 16#643D;
   // GBK_TO_UNICODE[16152] := 16#B2EC;
   // GBK_TO_UNICODE[16153] := 16#5BDF;
   // GBK_TO_UNICODE[16154] := 16#B2ED;
   // GBK_TO_UNICODE[16155] := 16#5C94;
   // GBK_TO_UNICODE[16156] := 16#B2EE;
   // GBK_TO_UNICODE[16157] := 16#5DEE;
   // GBK_TO_UNICODE[16158] := 16#B2EF;
   // GBK_TO_UNICODE[16159] := 16#8BE7;
   // GBK_TO_UNICODE[16160] := 16#B2F0;
   // GBK_TO_UNICODE[16161] := 16#62C6;
   // GBK_TO_UNICODE[16162] := 16#B2F1;
   // GBK_TO_UNICODE[16163] := 16#67F4;
   // GBK_TO_UNICODE[16164] := 16#B2F2;
   // GBK_TO_UNICODE[16165] := 16#8C7A;
   // GBK_TO_UNICODE[16166] := 16#B2F3;
   // GBK_TO_UNICODE[16167] := 16#6400;
   // GBK_TO_UNICODE[16168] := 16#B2F4;
   // GBK_TO_UNICODE[16169] := 16#63BA;
   // GBK_TO_UNICODE[16170] := 16#B2F5;
   // GBK_TO_UNICODE[16171] := 16#8749;
   // GBK_TO_UNICODE[16172] := 16#B2F6;
   // GBK_TO_UNICODE[16173] := 16#998B;
   // GBK_TO_UNICODE[16174] := 16#B2F7;
   // GBK_TO_UNICODE[16175] := 16#8C17;
   // GBK_TO_UNICODE[16176] := 16#B2F8;
   // GBK_TO_UNICODE[16177] := 16#7F20;
   // GBK_TO_UNICODE[16178] := 16#B2F9;
   // GBK_TO_UNICODE[16179] := 16#94F2;
   // GBK_TO_UNICODE[16180] := 16#B2FA;
   // GBK_TO_UNICODE[16181] := 16#4EA7;
   // GBK_TO_UNICODE[16182] := 16#B2FB;
   // GBK_TO_UNICODE[16183] := 16#9610;
   // GBK_TO_UNICODE[16184] := 16#B2FC;
   // GBK_TO_UNICODE[16185] := 16#98A4;
   // GBK_TO_UNICODE[16186] := 16#B2FD;
   // GBK_TO_UNICODE[16187] := 16#660C;
   // GBK_TO_UNICODE[16188] := 16#B2FE;
   // GBK_TO_UNICODE[16189] := 16#7316;
   // GBK_TO_UNICODE[16190] := 16#B340;
   // GBK_TO_UNICODE[16191] := 16#77E6;
   // GBK_TO_UNICODE[16192] := 16#B341;
   // GBK_TO_UNICODE[16193] := 16#77E8;
   // GBK_TO_UNICODE[16194] := 16#B342;
   // GBK_TO_UNICODE[16195] := 16#77EA;
   // GBK_TO_UNICODE[16196] := 16#B343;
   // GBK_TO_UNICODE[16197] := 16#77EF;
   // GBK_TO_UNICODE[16198] := 16#B344;
   // GBK_TO_UNICODE[16199] := 16#77F0;
   // GBK_TO_UNICODE[16200] := 16#B345;
   // GBK_TO_UNICODE[16201] := 16#77F1;
   // GBK_TO_UNICODE[16202] := 16#B346;
   // GBK_TO_UNICODE[16203] := 16#77F2;
   // GBK_TO_UNICODE[16204] := 16#B347;
   // GBK_TO_UNICODE[16205] := 16#77F4;
   // GBK_TO_UNICODE[16206] := 16#B348;
   // GBK_TO_UNICODE[16207] := 16#77F5;
   // GBK_TO_UNICODE[16208] := 16#B349;
   // GBK_TO_UNICODE[16209] := 16#77F7;
   // GBK_TO_UNICODE[16210] := 16#B34A;
   // GBK_TO_UNICODE[16211] := 16#77F9;
   // GBK_TO_UNICODE[16212] := 16#B34B;
   // GBK_TO_UNICODE[16213] := 16#77FA;
   // GBK_TO_UNICODE[16214] := 16#B34C;
   // GBK_TO_UNICODE[16215] := 16#77FB;
   // GBK_TO_UNICODE[16216] := 16#B34D;
   // GBK_TO_UNICODE[16217] := 16#77FC;
   // GBK_TO_UNICODE[16218] := 16#B34E;
   // GBK_TO_UNICODE[16219] := 16#7803;
   // GBK_TO_UNICODE[16220] := 16#B34F;
   // GBK_TO_UNICODE[16221] := 16#7804;
   // GBK_TO_UNICODE[16222] := 16#B350;
   // GBK_TO_UNICODE[16223] := 16#7805;
   // GBK_TO_UNICODE[16224] := 16#B351;
   // GBK_TO_UNICODE[16225] := 16#7806;
   // GBK_TO_UNICODE[16226] := 16#B352;
   // GBK_TO_UNICODE[16227] := 16#7807;
   // GBK_TO_UNICODE[16228] := 16#B353;
   // GBK_TO_UNICODE[16229] := 16#7808;
   // GBK_TO_UNICODE[16230] := 16#B354;
   // GBK_TO_UNICODE[16231] := 16#780A;
   // GBK_TO_UNICODE[16232] := 16#B355;
   // GBK_TO_UNICODE[16233] := 16#780B;
   // GBK_TO_UNICODE[16234] := 16#B356;
   // GBK_TO_UNICODE[16235] := 16#780E;
   // GBK_TO_UNICODE[16236] := 16#B357;
   // GBK_TO_UNICODE[16237] := 16#780F;
   // GBK_TO_UNICODE[16238] := 16#B358;
   // GBK_TO_UNICODE[16239] := 16#7810;
   // GBK_TO_UNICODE[16240] := 16#B359;
   // GBK_TO_UNICODE[16241] := 16#7813;
   // GBK_TO_UNICODE[16242] := 16#B35A;
   // GBK_TO_UNICODE[16243] := 16#7815;
   // GBK_TO_UNICODE[16244] := 16#B35B;
   // GBK_TO_UNICODE[16245] := 16#7819;
   // GBK_TO_UNICODE[16246] := 16#B35C;
   // GBK_TO_UNICODE[16247] := 16#781B;
   // GBK_TO_UNICODE[16248] := 16#B35D;
   // GBK_TO_UNICODE[16249] := 16#781E;
   // GBK_TO_UNICODE[16250] := 16#B35E;
   // GBK_TO_UNICODE[16251] := 16#7820;
   // GBK_TO_UNICODE[16252] := 16#B35F;
   // GBK_TO_UNICODE[16253] := 16#7821;
   // GBK_TO_UNICODE[16254] := 16#B360;
   // GBK_TO_UNICODE[16255] := 16#7822;
   // GBK_TO_UNICODE[16256] := 16#B361;
   // GBK_TO_UNICODE[16257] := 16#7824;
   // GBK_TO_UNICODE[16258] := 16#B362;
   // GBK_TO_UNICODE[16259] := 16#7828;
   // GBK_TO_UNICODE[16260] := 16#B363;
   // GBK_TO_UNICODE[16261] := 16#782A;
   // GBK_TO_UNICODE[16262] := 16#B364;
   // GBK_TO_UNICODE[16263] := 16#782B;
   // GBK_TO_UNICODE[16264] := 16#B365;
   // GBK_TO_UNICODE[16265] := 16#782E;
   // GBK_TO_UNICODE[16266] := 16#B366;
   // GBK_TO_UNICODE[16267] := 16#782F;
   // GBK_TO_UNICODE[16268] := 16#B367;
   // GBK_TO_UNICODE[16269] := 16#7831;
   // GBK_TO_UNICODE[16270] := 16#B368;
   // GBK_TO_UNICODE[16271] := 16#7832;
   // GBK_TO_UNICODE[16272] := 16#B369;
   // GBK_TO_UNICODE[16273] := 16#7833;
   // GBK_TO_UNICODE[16274] := 16#B36A;
   // GBK_TO_UNICODE[16275] := 16#7835;
   // GBK_TO_UNICODE[16276] := 16#B36B;
   // GBK_TO_UNICODE[16277] := 16#7836;
   // GBK_TO_UNICODE[16278] := 16#B36C;
   // GBK_TO_UNICODE[16279] := 16#783D;
   // GBK_TO_UNICODE[16280] := 16#B36D;
   // GBK_TO_UNICODE[16281] := 16#783F;
   // GBK_TO_UNICODE[16282] := 16#B36E;
   // GBK_TO_UNICODE[16283] := 16#7841;
   // GBK_TO_UNICODE[16284] := 16#B36F;
   // GBK_TO_UNICODE[16285] := 16#7842;
   // GBK_TO_UNICODE[16286] := 16#B370;
   // GBK_TO_UNICODE[16287] := 16#7843;
   // GBK_TO_UNICODE[16288] := 16#B371;
   // GBK_TO_UNICODE[16289] := 16#7844;
   // GBK_TO_UNICODE[16290] := 16#B372;
   // GBK_TO_UNICODE[16291] := 16#7846;
   // GBK_TO_UNICODE[16292] := 16#B373;
   // GBK_TO_UNICODE[16293] := 16#7848;
   // GBK_TO_UNICODE[16294] := 16#B374;
   // GBK_TO_UNICODE[16295] := 16#7849;
   // GBK_TO_UNICODE[16296] := 16#B375;
   // GBK_TO_UNICODE[16297] := 16#784A;
   // GBK_TO_UNICODE[16298] := 16#B376;
   // GBK_TO_UNICODE[16299] := 16#784B;
   // GBK_TO_UNICODE[16300] := 16#B377;
   // GBK_TO_UNICODE[16301] := 16#784D;
   // GBK_TO_UNICODE[16302] := 16#B378;
   // GBK_TO_UNICODE[16303] := 16#784F;
   // GBK_TO_UNICODE[16304] := 16#B379;
   // GBK_TO_UNICODE[16305] := 16#7851;
   // GBK_TO_UNICODE[16306] := 16#B37A;
   // GBK_TO_UNICODE[16307] := 16#7853;
   // GBK_TO_UNICODE[16308] := 16#B37B;
   // GBK_TO_UNICODE[16309] := 16#7854;
   // GBK_TO_UNICODE[16310] := 16#B37C;
   // GBK_TO_UNICODE[16311] := 16#7858;
   // GBK_TO_UNICODE[16312] := 16#B37D;
   // GBK_TO_UNICODE[16313] := 16#7859;
   // GBK_TO_UNICODE[16314] := 16#B37E;
   // GBK_TO_UNICODE[16315] := 16#785A;
   // GBK_TO_UNICODE[16316] := 16#B380;
   // GBK_TO_UNICODE[16317] := 16#785B;
   // GBK_TO_UNICODE[16318] := 16#B381;
   // GBK_TO_UNICODE[16319] := 16#785C;
   // GBK_TO_UNICODE[16320] := 16#B382;
   // GBK_TO_UNICODE[16321] := 16#785E;
   // GBK_TO_UNICODE[16322] := 16#B383;
   // GBK_TO_UNICODE[16323] := 16#785F;
   // GBK_TO_UNICODE[16324] := 16#B384;
   // GBK_TO_UNICODE[16325] := 16#7860;
   // GBK_TO_UNICODE[16326] := 16#B385;
   // GBK_TO_UNICODE[16327] := 16#7861;
   // GBK_TO_UNICODE[16328] := 16#B386;
   // GBK_TO_UNICODE[16329] := 16#7862;
   // GBK_TO_UNICODE[16330] := 16#B387;
   // GBK_TO_UNICODE[16331] := 16#7863;
   // GBK_TO_UNICODE[16332] := 16#B388;
   // GBK_TO_UNICODE[16333] := 16#7864;
   // GBK_TO_UNICODE[16334] := 16#B389;
   // GBK_TO_UNICODE[16335] := 16#7865;
   // GBK_TO_UNICODE[16336] := 16#B38A;
   // GBK_TO_UNICODE[16337] := 16#7866;
   // GBK_TO_UNICODE[16338] := 16#B38B;
   // GBK_TO_UNICODE[16339] := 16#7867;
   // GBK_TO_UNICODE[16340] := 16#B38C;
   // GBK_TO_UNICODE[16341] := 16#7868;
   // GBK_TO_UNICODE[16342] := 16#B38D;
   // GBK_TO_UNICODE[16343] := 16#7869;
   // GBK_TO_UNICODE[16344] := 16#B38E;
   // GBK_TO_UNICODE[16345] := 16#786F;
   // GBK_TO_UNICODE[16346] := 16#B38F;
   // GBK_TO_UNICODE[16347] := 16#7870;
   // GBK_TO_UNICODE[16348] := 16#B390;
   // GBK_TO_UNICODE[16349] := 16#7871;
   // GBK_TO_UNICODE[16350] := 16#B391;
   // GBK_TO_UNICODE[16351] := 16#7872;
   // GBK_TO_UNICODE[16352] := 16#B392;
   // GBK_TO_UNICODE[16353] := 16#7873;
   // GBK_TO_UNICODE[16354] := 16#B393;
   // GBK_TO_UNICODE[16355] := 16#7874;
   // GBK_TO_UNICODE[16356] := 16#B394;
   // GBK_TO_UNICODE[16357] := 16#7875;
   // GBK_TO_UNICODE[16358] := 16#B395;
   // GBK_TO_UNICODE[16359] := 16#7876;
   // GBK_TO_UNICODE[16360] := 16#B396;
   // GBK_TO_UNICODE[16361] := 16#7878;
   // GBK_TO_UNICODE[16362] := 16#B397;
   // GBK_TO_UNICODE[16363] := 16#7879;
   // GBK_TO_UNICODE[16364] := 16#B398;
   // GBK_TO_UNICODE[16365] := 16#787A;
   // GBK_TO_UNICODE[16366] := 16#B399;
   // GBK_TO_UNICODE[16367] := 16#787B;
   // GBK_TO_UNICODE[16368] := 16#B39A;
   // GBK_TO_UNICODE[16369] := 16#787D;
   // GBK_TO_UNICODE[16370] := 16#B39B;
   // GBK_TO_UNICODE[16371] := 16#787E;
   // GBK_TO_UNICODE[16372] := 16#B39C;
   // GBK_TO_UNICODE[16373] := 16#787F;
   // GBK_TO_UNICODE[16374] := 16#B39D;
   // GBK_TO_UNICODE[16375] := 16#7880;
   // GBK_TO_UNICODE[16376] := 16#B39E;
   // GBK_TO_UNICODE[16377] := 16#7881;
   // GBK_TO_UNICODE[16378] := 16#B39F;
   // GBK_TO_UNICODE[16379] := 16#7882;
   // GBK_TO_UNICODE[16380] := 16#B3A0;
   // GBK_TO_UNICODE[16381] := 16#7883;
   // GBK_TO_UNICODE[16382] := 16#B3A1;
   // GBK_TO_UNICODE[16383] := 16#573A;
   // GBK_TO_UNICODE[16384] := 16#B3A2;
   // GBK_TO_UNICODE[16385] := 16#5C1D;
   // GBK_TO_UNICODE[16386] := 16#B3A3;
   // GBK_TO_UNICODE[16387] := 16#5E38;
   // GBK_TO_UNICODE[16388] := 16#B3A4;
   // GBK_TO_UNICODE[16389] := 16#957F;
   // GBK_TO_UNICODE[16390] := 16#B3A5;
   // GBK_TO_UNICODE[16391] := 16#507F;
   // GBK_TO_UNICODE[16392] := 16#B3A6;
   // GBK_TO_UNICODE[16393] := 16#80A0;
   // GBK_TO_UNICODE[16394] := 16#B3A7;
   // GBK_TO_UNICODE[16395] := 16#5382;
   // GBK_TO_UNICODE[16396] := 16#B3A8;
   // GBK_TO_UNICODE[16397] := 16#655E;
   // GBK_TO_UNICODE[16398] := 16#B3A9;
   // GBK_TO_UNICODE[16399] := 16#7545;
   // GBK_TO_UNICODE[16400] := 16#B3AA;
   // GBK_TO_UNICODE[16401] := 16#5531;
   // GBK_TO_UNICODE[16402] := 16#B3AB;
   // GBK_TO_UNICODE[16403] := 16#5021;
   // GBK_TO_UNICODE[16404] := 16#B3AC;
   // GBK_TO_UNICODE[16405] := 16#8D85;
   // GBK_TO_UNICODE[16406] := 16#B3AD;
   // GBK_TO_UNICODE[16407] := 16#6284;
   // GBK_TO_UNICODE[16408] := 16#B3AE;
   // GBK_TO_UNICODE[16409] := 16#949E;
   // GBK_TO_UNICODE[16410] := 16#B3AF;
   // GBK_TO_UNICODE[16411] := 16#671D;
   // GBK_TO_UNICODE[16412] := 16#B3B0;
   // GBK_TO_UNICODE[16413] := 16#5632;
   // GBK_TO_UNICODE[16414] := 16#B3B1;
   // GBK_TO_UNICODE[16415] := 16#6F6E;
   // GBK_TO_UNICODE[16416] := 16#B3B2;
   // GBK_TO_UNICODE[16417] := 16#5DE2;
   // GBK_TO_UNICODE[16418] := 16#B3B3;
   // GBK_TO_UNICODE[16419] := 16#5435;
   // GBK_TO_UNICODE[16420] := 16#B3B4;
   // GBK_TO_UNICODE[16421] := 16#7092;
   // GBK_TO_UNICODE[16422] := 16#B3B5;
   // GBK_TO_UNICODE[16423] := 16#8F66;
   // GBK_TO_UNICODE[16424] := 16#B3B6;
   // GBK_TO_UNICODE[16425] := 16#626F;
   // GBK_TO_UNICODE[16426] := 16#B3B7;
   // GBK_TO_UNICODE[16427] := 16#64A4;
   // GBK_TO_UNICODE[16428] := 16#B3B8;
   // GBK_TO_UNICODE[16429] := 16#63A3;
   // GBK_TO_UNICODE[16430] := 16#B3B9;
   // GBK_TO_UNICODE[16431] := 16#5F7B;
   // GBK_TO_UNICODE[16432] := 16#B3BA;
   // GBK_TO_UNICODE[16433] := 16#6F88;
   // GBK_TO_UNICODE[16434] := 16#B3BB;
   // GBK_TO_UNICODE[16435] := 16#90F4;
   // GBK_TO_UNICODE[16436] := 16#B3BC;
   // GBK_TO_UNICODE[16437] := 16#81E3;
   // GBK_TO_UNICODE[16438] := 16#B3BD;
   // GBK_TO_UNICODE[16439] := 16#8FB0;
   // GBK_TO_UNICODE[16440] := 16#B3BE;
   // GBK_TO_UNICODE[16441] := 16#5C18;
   // GBK_TO_UNICODE[16442] := 16#B3BF;
   // GBK_TO_UNICODE[16443] := 16#6668;
   // GBK_TO_UNICODE[16444] := 16#B3C0;
   // GBK_TO_UNICODE[16445] := 16#5FF1;
   // GBK_TO_UNICODE[16446] := 16#B3C1;
   // GBK_TO_UNICODE[16447] := 16#6C89;
   // GBK_TO_UNICODE[16448] := 16#B3C2;
   // GBK_TO_UNICODE[16449] := 16#9648;
   // GBK_TO_UNICODE[16450] := 16#B3C3;
   // GBK_TO_UNICODE[16451] := 16#8D81;
   // GBK_TO_UNICODE[16452] := 16#B3C4;
   // GBK_TO_UNICODE[16453] := 16#886C;
   // GBK_TO_UNICODE[16454] := 16#B3C5;
   // GBK_TO_UNICODE[16455] := 16#6491;
   // GBK_TO_UNICODE[16456] := 16#B3C6;
   // GBK_TO_UNICODE[16457] := 16#79F0;
   // GBK_TO_UNICODE[16458] := 16#B3C7;
   // GBK_TO_UNICODE[16459] := 16#57CE;
   // GBK_TO_UNICODE[16460] := 16#B3C8;
   // GBK_TO_UNICODE[16461] := 16#6A59;
   // GBK_TO_UNICODE[16462] := 16#B3C9;
   // GBK_TO_UNICODE[16463] := 16#6210;
   // GBK_TO_UNICODE[16464] := 16#B3CA;
   // GBK_TO_UNICODE[16465] := 16#5448;
   // GBK_TO_UNICODE[16466] := 16#B3CB;
   // GBK_TO_UNICODE[16467] := 16#4E58;
   // GBK_TO_UNICODE[16468] := 16#B3CC;
   // GBK_TO_UNICODE[16469] := 16#7A0B;
   // GBK_TO_UNICODE[16470] := 16#B3CD;
   // GBK_TO_UNICODE[16471] := 16#60E9;
   // GBK_TO_UNICODE[16472] := 16#B3CE;
   // GBK_TO_UNICODE[16473] := 16#6F84;
   // GBK_TO_UNICODE[16474] := 16#B3CF;
   // GBK_TO_UNICODE[16475] := 16#8BDA;
   // GBK_TO_UNICODE[16476] := 16#B3D0;
   // GBK_TO_UNICODE[16477] := 16#627F;
   // GBK_TO_UNICODE[16478] := 16#B3D1;
   // GBK_TO_UNICODE[16479] := 16#901E;
   // GBK_TO_UNICODE[16480] := 16#B3D2;
   // GBK_TO_UNICODE[16481] := 16#9A8B;
   // GBK_TO_UNICODE[16482] := 16#B3D3;
   // GBK_TO_UNICODE[16483] := 16#79E4;
   // GBK_TO_UNICODE[16484] := 16#B3D4;
   // GBK_TO_UNICODE[16485] := 16#5403;
   // GBK_TO_UNICODE[16486] := 16#B3D5;
   // GBK_TO_UNICODE[16487] := 16#75F4;
   // GBK_TO_UNICODE[16488] := 16#B3D6;
   // GBK_TO_UNICODE[16489] := 16#6301;
   // GBK_TO_UNICODE[16490] := 16#B3D7;
   // GBK_TO_UNICODE[16491] := 16#5319;
   // GBK_TO_UNICODE[16492] := 16#B3D8;
   // GBK_TO_UNICODE[16493] := 16#6C60;
   // GBK_TO_UNICODE[16494] := 16#B3D9;
   // GBK_TO_UNICODE[16495] := 16#8FDF;
   // GBK_TO_UNICODE[16496] := 16#B3DA;
   // GBK_TO_UNICODE[16497] := 16#5F1B;
   // GBK_TO_UNICODE[16498] := 16#B3DB;
   // GBK_TO_UNICODE[16499] := 16#9A70;
   // GBK_TO_UNICODE[16500] := 16#B3DC;
   // GBK_TO_UNICODE[16501] := 16#803B;
   // GBK_TO_UNICODE[16502] := 16#B3DD;
   // GBK_TO_UNICODE[16503] := 16#9F7F;
   // GBK_TO_UNICODE[16504] := 16#B3DE;
   // GBK_TO_UNICODE[16505] := 16#4F88;
   // GBK_TO_UNICODE[16506] := 16#B3DF;
   // GBK_TO_UNICODE[16507] := 16#5C3A;
   // GBK_TO_UNICODE[16508] := 16#B3E0;
   // GBK_TO_UNICODE[16509] := 16#8D64;
   // GBK_TO_UNICODE[16510] := 16#B3E1;
   // GBK_TO_UNICODE[16511] := 16#7FC5;
   // GBK_TO_UNICODE[16512] := 16#B3E2;
   // GBK_TO_UNICODE[16513] := 16#65A5;
   // GBK_TO_UNICODE[16514] := 16#B3E3;
   // GBK_TO_UNICODE[16515] := 16#70BD;
   // GBK_TO_UNICODE[16516] := 16#B3E4;
   // GBK_TO_UNICODE[16517] := 16#5145;
   // GBK_TO_UNICODE[16518] := 16#B3E5;
   // GBK_TO_UNICODE[16519] := 16#51B2;
   // GBK_TO_UNICODE[16520] := 16#B3E6;
   // GBK_TO_UNICODE[16521] := 16#866B;
   // GBK_TO_UNICODE[16522] := 16#B3E7;
   // GBK_TO_UNICODE[16523] := 16#5D07;
   // GBK_TO_UNICODE[16524] := 16#B3E8;
   // GBK_TO_UNICODE[16525] := 16#5BA0;
   // GBK_TO_UNICODE[16526] := 16#B3E9;
   // GBK_TO_UNICODE[16527] := 16#62BD;
   // GBK_TO_UNICODE[16528] := 16#B3EA;
   // GBK_TO_UNICODE[16529] := 16#916C;
   // GBK_TO_UNICODE[16530] := 16#B3EB;
   // GBK_TO_UNICODE[16531] := 16#7574;
   // GBK_TO_UNICODE[16532] := 16#B3EC;
   // GBK_TO_UNICODE[16533] := 16#8E0C;
   // GBK_TO_UNICODE[16534] := 16#B3ED;
   // GBK_TO_UNICODE[16535] := 16#7A20;
   // GBK_TO_UNICODE[16536] := 16#B3EE;
   // GBK_TO_UNICODE[16537] := 16#6101;
   // GBK_TO_UNICODE[16538] := 16#B3EF;
   // GBK_TO_UNICODE[16539] := 16#7B79;
   // GBK_TO_UNICODE[16540] := 16#B3F0;
   // GBK_TO_UNICODE[16541] := 16#4EC7;
   // GBK_TO_UNICODE[16542] := 16#B3F1;
   // GBK_TO_UNICODE[16543] := 16#7EF8;
   // GBK_TO_UNICODE[16544] := 16#B3F2;
   // GBK_TO_UNICODE[16545] := 16#7785;
   // GBK_TO_UNICODE[16546] := 16#B3F3;
   // GBK_TO_UNICODE[16547] := 16#4E11;
   // GBK_TO_UNICODE[16548] := 16#B3F4;
   // GBK_TO_UNICODE[16549] := 16#81ED;
   // GBK_TO_UNICODE[16550] := 16#B3F5;
   // GBK_TO_UNICODE[16551] := 16#521D;
   // GBK_TO_UNICODE[16552] := 16#B3F6;
   // GBK_TO_UNICODE[16553] := 16#51FA;
   // GBK_TO_UNICODE[16554] := 16#B3F7;
   // GBK_TO_UNICODE[16555] := 16#6A71;
   // GBK_TO_UNICODE[16556] := 16#B3F8;
   // GBK_TO_UNICODE[16557] := 16#53A8;
   // GBK_TO_UNICODE[16558] := 16#B3F9;
   // GBK_TO_UNICODE[16559] := 16#8E87;
   // GBK_TO_UNICODE[16560] := 16#B3FA;
   // GBK_TO_UNICODE[16561] := 16#9504;
   // GBK_TO_UNICODE[16562] := 16#B3FB;
   // GBK_TO_UNICODE[16563] := 16#96CF;
   // GBK_TO_UNICODE[16564] := 16#B3FC;
   // GBK_TO_UNICODE[16565] := 16#6EC1;
   // GBK_TO_UNICODE[16566] := 16#B3FD;
   // GBK_TO_UNICODE[16567] := 16#9664;
   // GBK_TO_UNICODE[16568] := 16#B3FE;
   // GBK_TO_UNICODE[16569] := 16#695A;
   // GBK_TO_UNICODE[16570] := 16#B440;
   // GBK_TO_UNICODE[16571] := 16#7884;
   // GBK_TO_UNICODE[16572] := 16#B441;
   // GBK_TO_UNICODE[16573] := 16#7885;
   // GBK_TO_UNICODE[16574] := 16#B442;
   // GBK_TO_UNICODE[16575] := 16#7886;
   // GBK_TO_UNICODE[16576] := 16#B443;
   // GBK_TO_UNICODE[16577] := 16#7888;
   // GBK_TO_UNICODE[16578] := 16#B444;
   // GBK_TO_UNICODE[16579] := 16#788A;
   // GBK_TO_UNICODE[16580] := 16#B445;
   // GBK_TO_UNICODE[16581] := 16#788B;
   // GBK_TO_UNICODE[16582] := 16#B446;
   // GBK_TO_UNICODE[16583] := 16#788F;
   // GBK_TO_UNICODE[16584] := 16#B447;
   // GBK_TO_UNICODE[16585] := 16#7890;
   // GBK_TO_UNICODE[16586] := 16#B448;
   // GBK_TO_UNICODE[16587] := 16#7892;
   // GBK_TO_UNICODE[16588] := 16#B449;
   // GBK_TO_UNICODE[16589] := 16#7894;
   // GBK_TO_UNICODE[16590] := 16#B44A;
   // GBK_TO_UNICODE[16591] := 16#7895;
   // GBK_TO_UNICODE[16592] := 16#B44B;
   // GBK_TO_UNICODE[16593] := 16#7896;
   // GBK_TO_UNICODE[16594] := 16#B44C;
   // GBK_TO_UNICODE[16595] := 16#7899;
   // GBK_TO_UNICODE[16596] := 16#B44D;
   // GBK_TO_UNICODE[16597] := 16#789D;
   // GBK_TO_UNICODE[16598] := 16#B44E;
   // GBK_TO_UNICODE[16599] := 16#789E;
   // GBK_TO_UNICODE[16600] := 16#B44F;
   // GBK_TO_UNICODE[16601] := 16#78A0;
   // GBK_TO_UNICODE[16602] := 16#B450;
   // GBK_TO_UNICODE[16603] := 16#78A2;
   // GBK_TO_UNICODE[16604] := 16#B451;
   // GBK_TO_UNICODE[16605] := 16#78A4;
   // GBK_TO_UNICODE[16606] := 16#B452;
   // GBK_TO_UNICODE[16607] := 16#78A6;
   // GBK_TO_UNICODE[16608] := 16#B453;
   // GBK_TO_UNICODE[16609] := 16#78A8;
   // GBK_TO_UNICODE[16610] := 16#B454;
   // GBK_TO_UNICODE[16611] := 16#78A9;
   // GBK_TO_UNICODE[16612] := 16#B455;
   // GBK_TO_UNICODE[16613] := 16#78AA;
   // GBK_TO_UNICODE[16614] := 16#B456;
   // GBK_TO_UNICODE[16615] := 16#78AB;
   // GBK_TO_UNICODE[16616] := 16#B457;
   // GBK_TO_UNICODE[16617] := 16#78AC;
   // GBK_TO_UNICODE[16618] := 16#B458;
   // GBK_TO_UNICODE[16619] := 16#78AD;
   // GBK_TO_UNICODE[16620] := 16#B459;
   // GBK_TO_UNICODE[16621] := 16#78AE;
   // GBK_TO_UNICODE[16622] := 16#B45A;
   // GBK_TO_UNICODE[16623] := 16#78AF;
   // GBK_TO_UNICODE[16624] := 16#B45B;
   // GBK_TO_UNICODE[16625] := 16#78B5;
   // GBK_TO_UNICODE[16626] := 16#B45C;
   // GBK_TO_UNICODE[16627] := 16#78B6;
   // GBK_TO_UNICODE[16628] := 16#B45D;
   // GBK_TO_UNICODE[16629] := 16#78B7;
   // GBK_TO_UNICODE[16630] := 16#B45E;
   // GBK_TO_UNICODE[16631] := 16#78B8;
   // GBK_TO_UNICODE[16632] := 16#B45F;
   // GBK_TO_UNICODE[16633] := 16#78BA;
   // GBK_TO_UNICODE[16634] := 16#B460;
   // GBK_TO_UNICODE[16635] := 16#78BB;
   // GBK_TO_UNICODE[16636] := 16#B461;
   // GBK_TO_UNICODE[16637] := 16#78BC;
   // GBK_TO_UNICODE[16638] := 16#B462;
   // GBK_TO_UNICODE[16639] := 16#78BD;
   // GBK_TO_UNICODE[16640] := 16#B463;
   // GBK_TO_UNICODE[16641] := 16#78BF;
   // GBK_TO_UNICODE[16642] := 16#B464;
   // GBK_TO_UNICODE[16643] := 16#78C0;
   // GBK_TO_UNICODE[16644] := 16#B465;
   // GBK_TO_UNICODE[16645] := 16#78C2;
   // GBK_TO_UNICODE[16646] := 16#B466;
   // GBK_TO_UNICODE[16647] := 16#78C3;
   // GBK_TO_UNICODE[16648] := 16#B467;
   // GBK_TO_UNICODE[16649] := 16#78C4;
   // GBK_TO_UNICODE[16650] := 16#B468;
   // GBK_TO_UNICODE[16651] := 16#78C6;
   // GBK_TO_UNICODE[16652] := 16#B469;
   // GBK_TO_UNICODE[16653] := 16#78C7;
   // GBK_TO_UNICODE[16654] := 16#B46A;
   // GBK_TO_UNICODE[16655] := 16#78C8;
   // GBK_TO_UNICODE[16656] := 16#B46B;
   // GBK_TO_UNICODE[16657] := 16#78CC;
   // GBK_TO_UNICODE[16658] := 16#B46C;
   // GBK_TO_UNICODE[16659] := 16#78CD;
   // GBK_TO_UNICODE[16660] := 16#B46D;
   // GBK_TO_UNICODE[16661] := 16#78CE;
   // GBK_TO_UNICODE[16662] := 16#B46E;
   // GBK_TO_UNICODE[16663] := 16#78CF;
   // GBK_TO_UNICODE[16664] := 16#B46F;
   // GBK_TO_UNICODE[16665] := 16#78D1;
   // GBK_TO_UNICODE[16666] := 16#B470;
   // GBK_TO_UNICODE[16667] := 16#78D2;
   // GBK_TO_UNICODE[16668] := 16#B471;
   // GBK_TO_UNICODE[16669] := 16#78D3;
   // GBK_TO_UNICODE[16670] := 16#B472;
   // GBK_TO_UNICODE[16671] := 16#78D6;
   // GBK_TO_UNICODE[16672] := 16#B473;
   // GBK_TO_UNICODE[16673] := 16#78D7;
   // GBK_TO_UNICODE[16674] := 16#B474;
   // GBK_TO_UNICODE[16675] := 16#78D8;
   // GBK_TO_UNICODE[16676] := 16#B475;
   // GBK_TO_UNICODE[16677] := 16#78DA;
   // GBK_TO_UNICODE[16678] := 16#B476;
   // GBK_TO_UNICODE[16679] := 16#78DB;
   // GBK_TO_UNICODE[16680] := 16#B477;
   // GBK_TO_UNICODE[16681] := 16#78DC;
   // GBK_TO_UNICODE[16682] := 16#B478;
   // GBK_TO_UNICODE[16683] := 16#78DD;
   // GBK_TO_UNICODE[16684] := 16#B479;
   // GBK_TO_UNICODE[16685] := 16#78DE;
   // GBK_TO_UNICODE[16686] := 16#B47A;
   // GBK_TO_UNICODE[16687] := 16#78DF;
   // GBK_TO_UNICODE[16688] := 16#B47B;
   // GBK_TO_UNICODE[16689] := 16#78E0;
   // GBK_TO_UNICODE[16690] := 16#B47C;
   // GBK_TO_UNICODE[16691] := 16#78E1;
   // GBK_TO_UNICODE[16692] := 16#B47D;
   // GBK_TO_UNICODE[16693] := 16#78E2;
   // GBK_TO_UNICODE[16694] := 16#B47E;
   // GBK_TO_UNICODE[16695] := 16#78E3;
   // GBK_TO_UNICODE[16696] := 16#B480;
   // GBK_TO_UNICODE[16697] := 16#78E4;
   // GBK_TO_UNICODE[16698] := 16#B481;
   // GBK_TO_UNICODE[16699] := 16#78E5;
   // GBK_TO_UNICODE[16700] := 16#B482;
   // GBK_TO_UNICODE[16701] := 16#78E6;
   // GBK_TO_UNICODE[16702] := 16#B483;
   // GBK_TO_UNICODE[16703] := 16#78E7;
   // GBK_TO_UNICODE[16704] := 16#B484;
   // GBK_TO_UNICODE[16705] := 16#78E9;
   // GBK_TO_UNICODE[16706] := 16#B485;
   // GBK_TO_UNICODE[16707] := 16#78EA;
   // GBK_TO_UNICODE[16708] := 16#B486;
   // GBK_TO_UNICODE[16709] := 16#78EB;
   // GBK_TO_UNICODE[16710] := 16#B487;
   // GBK_TO_UNICODE[16711] := 16#78ED;
   // GBK_TO_UNICODE[16712] := 16#B488;
   // GBK_TO_UNICODE[16713] := 16#78EE;
   // GBK_TO_UNICODE[16714] := 16#B489;
   // GBK_TO_UNICODE[16715] := 16#78EF;
   // GBK_TO_UNICODE[16716] := 16#B48A;
   // GBK_TO_UNICODE[16717] := 16#78F0;
   // GBK_TO_UNICODE[16718] := 16#B48B;
   // GBK_TO_UNICODE[16719] := 16#78F1;
   // GBK_TO_UNICODE[16720] := 16#B48C;
   // GBK_TO_UNICODE[16721] := 16#78F3;
   // GBK_TO_UNICODE[16722] := 16#B48D;
   // GBK_TO_UNICODE[16723] := 16#78F5;
   // GBK_TO_UNICODE[16724] := 16#B48E;
   // GBK_TO_UNICODE[16725] := 16#78F6;
   // GBK_TO_UNICODE[16726] := 16#B48F;
   // GBK_TO_UNICODE[16727] := 16#78F8;
   // GBK_TO_UNICODE[16728] := 16#B490;
   // GBK_TO_UNICODE[16729] := 16#78F9;
   // GBK_TO_UNICODE[16730] := 16#B491;
   // GBK_TO_UNICODE[16731] := 16#78FB;
   // GBK_TO_UNICODE[16732] := 16#B492;
   // GBK_TO_UNICODE[16733] := 16#78FC;
   // GBK_TO_UNICODE[16734] := 16#B493;
   // GBK_TO_UNICODE[16735] := 16#78FD;
   // GBK_TO_UNICODE[16736] := 16#B494;
   // GBK_TO_UNICODE[16737] := 16#78FE;
   // GBK_TO_UNICODE[16738] := 16#B495;
   // GBK_TO_UNICODE[16739] := 16#78FF;
   // GBK_TO_UNICODE[16740] := 16#B496;
   // GBK_TO_UNICODE[16741] := 16#7900;
   // GBK_TO_UNICODE[16742] := 16#B497;
   // GBK_TO_UNICODE[16743] := 16#7902;
   // GBK_TO_UNICODE[16744] := 16#B498;
   // GBK_TO_UNICODE[16745] := 16#7903;
   // GBK_TO_UNICODE[16746] := 16#B499;
   // GBK_TO_UNICODE[16747] := 16#7904;
   // GBK_TO_UNICODE[16748] := 16#B49A;
   // GBK_TO_UNICODE[16749] := 16#7906;
   // GBK_TO_UNICODE[16750] := 16#B49B;
   // GBK_TO_UNICODE[16751] := 16#7907;
   // GBK_TO_UNICODE[16752] := 16#B49C;
   // GBK_TO_UNICODE[16753] := 16#7908;
   // GBK_TO_UNICODE[16754] := 16#B49D;
   // GBK_TO_UNICODE[16755] := 16#7909;
   // GBK_TO_UNICODE[16756] := 16#B49E;
   // GBK_TO_UNICODE[16757] := 16#790A;
   // GBK_TO_UNICODE[16758] := 16#B49F;
   // GBK_TO_UNICODE[16759] := 16#790B;
   // GBK_TO_UNICODE[16760] := 16#B4A0;
   // GBK_TO_UNICODE[16761] := 16#790C;
   // GBK_TO_UNICODE[16762] := 16#B4A1;
   // GBK_TO_UNICODE[16763] := 16#7840;
   // GBK_TO_UNICODE[16764] := 16#B4A2;
   // GBK_TO_UNICODE[16765] := 16#50A8;
   // GBK_TO_UNICODE[16766] := 16#B4A3;
   // GBK_TO_UNICODE[16767] := 16#77D7;
   // GBK_TO_UNICODE[16768] := 16#B4A4;
   // GBK_TO_UNICODE[16769] := 16#6410;
   // GBK_TO_UNICODE[16770] := 16#B4A5;
   // GBK_TO_UNICODE[16771] := 16#89E6;
   // GBK_TO_UNICODE[16772] := 16#B4A6;
   // GBK_TO_UNICODE[16773] := 16#5904;
   // GBK_TO_UNICODE[16774] := 16#B4A7;
   // GBK_TO_UNICODE[16775] := 16#63E3;
   // GBK_TO_UNICODE[16776] := 16#B4A8;
   // GBK_TO_UNICODE[16777] := 16#5DDD;
   // GBK_TO_UNICODE[16778] := 16#B4A9;
   // GBK_TO_UNICODE[16779] := 16#7A7F;
   // GBK_TO_UNICODE[16780] := 16#B4AA;
   // GBK_TO_UNICODE[16781] := 16#693D;
   // GBK_TO_UNICODE[16782] := 16#B4AB;
   // GBK_TO_UNICODE[16783] := 16#4F20;
   // GBK_TO_UNICODE[16784] := 16#B4AC;
   // GBK_TO_UNICODE[16785] := 16#8239;
   // GBK_TO_UNICODE[16786] := 16#B4AD;
   // GBK_TO_UNICODE[16787] := 16#5598;
   // GBK_TO_UNICODE[16788] := 16#B4AE;
   // GBK_TO_UNICODE[16789] := 16#4E32;
   // GBK_TO_UNICODE[16790] := 16#B4AF;
   // GBK_TO_UNICODE[16791] := 16#75AE;
   // GBK_TO_UNICODE[16792] := 16#B4B0;
   // GBK_TO_UNICODE[16793] := 16#7A97;
   // GBK_TO_UNICODE[16794] := 16#B4B1;
   // GBK_TO_UNICODE[16795] := 16#5E62;
   // GBK_TO_UNICODE[16796] := 16#B4B2;
   // GBK_TO_UNICODE[16797] := 16#5E8A;
   // GBK_TO_UNICODE[16798] := 16#B4B3;
   // GBK_TO_UNICODE[16799] := 16#95EF;
   // GBK_TO_UNICODE[16800] := 16#B4B4;
   // GBK_TO_UNICODE[16801] := 16#521B;
   // GBK_TO_UNICODE[16802] := 16#B4B5;
   // GBK_TO_UNICODE[16803] := 16#5439;
   // GBK_TO_UNICODE[16804] := 16#B4B6;
   // GBK_TO_UNICODE[16805] := 16#708A;
   // GBK_TO_UNICODE[16806] := 16#B4B7;
   // GBK_TO_UNICODE[16807] := 16#6376;
   // GBK_TO_UNICODE[16808] := 16#B4B8;
   // GBK_TO_UNICODE[16809] := 16#9524;
   // GBK_TO_UNICODE[16810] := 16#B4B9;
   // GBK_TO_UNICODE[16811] := 16#5782;
   // GBK_TO_UNICODE[16812] := 16#B4BA;
   // GBK_TO_UNICODE[16813] := 16#6625;
   // GBK_TO_UNICODE[16814] := 16#B4BB;
   // GBK_TO_UNICODE[16815] := 16#693F;
   // GBK_TO_UNICODE[16816] := 16#B4BC;
   // GBK_TO_UNICODE[16817] := 16#9187;
   // GBK_TO_UNICODE[16818] := 16#B4BD;
   // GBK_TO_UNICODE[16819] := 16#5507;
   // GBK_TO_UNICODE[16820] := 16#B4BE;
   // GBK_TO_UNICODE[16821] := 16#6DF3;
   // GBK_TO_UNICODE[16822] := 16#B4BF;
   // GBK_TO_UNICODE[16823] := 16#7EAF;
   // GBK_TO_UNICODE[16824] := 16#B4C0;
   // GBK_TO_UNICODE[16825] := 16#8822;
   // GBK_TO_UNICODE[16826] := 16#B4C1;
   // GBK_TO_UNICODE[16827] := 16#6233;
   // GBK_TO_UNICODE[16828] := 16#B4C2;
   // GBK_TO_UNICODE[16829] := 16#7EF0;
   // GBK_TO_UNICODE[16830] := 16#B4C3;
   // GBK_TO_UNICODE[16831] := 16#75B5;
   // GBK_TO_UNICODE[16832] := 16#B4C4;
   // GBK_TO_UNICODE[16833] := 16#8328;
   // GBK_TO_UNICODE[16834] := 16#B4C5;
   // GBK_TO_UNICODE[16835] := 16#78C1;
   // GBK_TO_UNICODE[16836] := 16#B4C6;
   // GBK_TO_UNICODE[16837] := 16#96CC;
   // GBK_TO_UNICODE[16838] := 16#B4C7;
   // GBK_TO_UNICODE[16839] := 16#8F9E;
   // GBK_TO_UNICODE[16840] := 16#B4C8;
   // GBK_TO_UNICODE[16841] := 16#6148;
   // GBK_TO_UNICODE[16842] := 16#B4C9;
   // GBK_TO_UNICODE[16843] := 16#74F7;
   // GBK_TO_UNICODE[16844] := 16#B4CA;
   // GBK_TO_UNICODE[16845] := 16#8BCD;
   // GBK_TO_UNICODE[16846] := 16#B4CB;
   // GBK_TO_UNICODE[16847] := 16#6B64;
   // GBK_TO_UNICODE[16848] := 16#B4CC;
   // GBK_TO_UNICODE[16849] := 16#523A;
   // GBK_TO_UNICODE[16850] := 16#B4CD;
   // GBK_TO_UNICODE[16851] := 16#8D50;
   // GBK_TO_UNICODE[16852] := 16#B4CE;
   // GBK_TO_UNICODE[16853] := 16#6B21;
   // GBK_TO_UNICODE[16854] := 16#B4CF;
   // GBK_TO_UNICODE[16855] := 16#806A;
   // GBK_TO_UNICODE[16856] := 16#B4D0;
   // GBK_TO_UNICODE[16857] := 16#8471;
   // GBK_TO_UNICODE[16858] := 16#B4D1;
   // GBK_TO_UNICODE[16859] := 16#56F1;
   // GBK_TO_UNICODE[16860] := 16#B4D2;
   // GBK_TO_UNICODE[16861] := 16#5306;
   // GBK_TO_UNICODE[16862] := 16#B4D3;
   // GBK_TO_UNICODE[16863] := 16#4ECE;
   // GBK_TO_UNICODE[16864] := 16#B4D4;
   // GBK_TO_UNICODE[16865] := 16#4E1B;
   // GBK_TO_UNICODE[16866] := 16#B4D5;
   // GBK_TO_UNICODE[16867] := 16#51D1;
   // GBK_TO_UNICODE[16868] := 16#B4D6;
   // GBK_TO_UNICODE[16869] := 16#7C97;
   // GBK_TO_UNICODE[16870] := 16#B4D7;
   // GBK_TO_UNICODE[16871] := 16#918B;
   // GBK_TO_UNICODE[16872] := 16#B4D8;
   // GBK_TO_UNICODE[16873] := 16#7C07;
   // GBK_TO_UNICODE[16874] := 16#B4D9;
   // GBK_TO_UNICODE[16875] := 16#4FC3;
   // GBK_TO_UNICODE[16876] := 16#B4DA;
   // GBK_TO_UNICODE[16877] := 16#8E7F;
   // GBK_TO_UNICODE[16878] := 16#B4DB;
   // GBK_TO_UNICODE[16879] := 16#7BE1;
   // GBK_TO_UNICODE[16880] := 16#B4DC;
   // GBK_TO_UNICODE[16881] := 16#7A9C;
   // GBK_TO_UNICODE[16882] := 16#B4DD;
   // GBK_TO_UNICODE[16883] := 16#6467;
   // GBK_TO_UNICODE[16884] := 16#B4DE;
   // GBK_TO_UNICODE[16885] := 16#5D14;
   // GBK_TO_UNICODE[16886] := 16#B4DF;
   // GBK_TO_UNICODE[16887] := 16#50AC;
   // GBK_TO_UNICODE[16888] := 16#B4E0;
   // GBK_TO_UNICODE[16889] := 16#8106;
   // GBK_TO_UNICODE[16890] := 16#B4E1;
   // GBK_TO_UNICODE[16891] := 16#7601;
   // GBK_TO_UNICODE[16892] := 16#B4E2;
   // GBK_TO_UNICODE[16893] := 16#7CB9;
   // GBK_TO_UNICODE[16894] := 16#B4E3;
   // GBK_TO_UNICODE[16895] := 16#6DEC;
   // GBK_TO_UNICODE[16896] := 16#B4E4;
   // GBK_TO_UNICODE[16897] := 16#7FE0;
   // GBK_TO_UNICODE[16898] := 16#B4E5;
   // GBK_TO_UNICODE[16899] := 16#6751;
   // GBK_TO_UNICODE[16900] := 16#B4E6;
   // GBK_TO_UNICODE[16901] := 16#5B58;
   // GBK_TO_UNICODE[16902] := 16#B4E7;
   // GBK_TO_UNICODE[16903] := 16#5BF8;
   // GBK_TO_UNICODE[16904] := 16#B4E8;
   // GBK_TO_UNICODE[16905] := 16#78CB;
   // GBK_TO_UNICODE[16906] := 16#B4E9;
   // GBK_TO_UNICODE[16907] := 16#64AE;
   // GBK_TO_UNICODE[16908] := 16#B4EA;
   // GBK_TO_UNICODE[16909] := 16#6413;
   // GBK_TO_UNICODE[16910] := 16#B4EB;
   // GBK_TO_UNICODE[16911] := 16#63AA;
   // GBK_TO_UNICODE[16912] := 16#B4EC;
   // GBK_TO_UNICODE[16913] := 16#632B;
   // GBK_TO_UNICODE[16914] := 16#B4ED;
   // GBK_TO_UNICODE[16915] := 16#9519;
   // GBK_TO_UNICODE[16916] := 16#B4EE;
   // GBK_TO_UNICODE[16917] := 16#642D;
   // GBK_TO_UNICODE[16918] := 16#B4EF;
   // GBK_TO_UNICODE[16919] := 16#8FBE;
   // GBK_TO_UNICODE[16920] := 16#B4F0;
   // GBK_TO_UNICODE[16921] := 16#7B54;
   // GBK_TO_UNICODE[16922] := 16#B4F1;
   // GBK_TO_UNICODE[16923] := 16#7629;
   // GBK_TO_UNICODE[16924] := 16#B4F2;
   // GBK_TO_UNICODE[16925] := 16#6253;
   // GBK_TO_UNICODE[16926] := 16#B4F3;
   // GBK_TO_UNICODE[16927] := 16#5927;
   // GBK_TO_UNICODE[16928] := 16#B4F4;
   // GBK_TO_UNICODE[16929] := 16#5446;
   // GBK_TO_UNICODE[16930] := 16#B4F5;
   // GBK_TO_UNICODE[16931] := 16#6B79;
   // GBK_TO_UNICODE[16932] := 16#B4F6;
   // GBK_TO_UNICODE[16933] := 16#50A3;
   // GBK_TO_UNICODE[16934] := 16#B4F7;
   // GBK_TO_UNICODE[16935] := 16#6234;
   // GBK_TO_UNICODE[16936] := 16#B4F8;
   // GBK_TO_UNICODE[16937] := 16#5E26;
   // GBK_TO_UNICODE[16938] := 16#B4F9;
   // GBK_TO_UNICODE[16939] := 16#6B86;
   // GBK_TO_UNICODE[16940] := 16#B4FA;
   // GBK_TO_UNICODE[16941] := 16#4EE3;
   // GBK_TO_UNICODE[16942] := 16#B4FB;
   // GBK_TO_UNICODE[16943] := 16#8D37;
   // GBK_TO_UNICODE[16944] := 16#B4FC;
   // GBK_TO_UNICODE[16945] := 16#888B;
   // GBK_TO_UNICODE[16946] := 16#B4FD;
   // GBK_TO_UNICODE[16947] := 16#5F85;
   // GBK_TO_UNICODE[16948] := 16#B4FE;
   // GBK_TO_UNICODE[16949] := 16#902E;
   // GBK_TO_UNICODE[16950] := 16#B540;
   // GBK_TO_UNICODE[16951] := 16#790D;
   // GBK_TO_UNICODE[16952] := 16#B541;
   // GBK_TO_UNICODE[16953] := 16#790E;
   // GBK_TO_UNICODE[16954] := 16#B542;
   // GBK_TO_UNICODE[16955] := 16#790F;
   // GBK_TO_UNICODE[16956] := 16#B543;
   // GBK_TO_UNICODE[16957] := 16#7910;
   // GBK_TO_UNICODE[16958] := 16#B544;
   // GBK_TO_UNICODE[16959] := 16#7911;
   // GBK_TO_UNICODE[16960] := 16#B545;
   // GBK_TO_UNICODE[16961] := 16#7912;
   // GBK_TO_UNICODE[16962] := 16#B546;
   // GBK_TO_UNICODE[16963] := 16#7914;
   // GBK_TO_UNICODE[16964] := 16#B547;
   // GBK_TO_UNICODE[16965] := 16#7915;
   // GBK_TO_UNICODE[16966] := 16#B548;
   // GBK_TO_UNICODE[16967] := 16#7916;
   // GBK_TO_UNICODE[16968] := 16#B549;
   // GBK_TO_UNICODE[16969] := 16#7917;
   // GBK_TO_UNICODE[16970] := 16#B54A;
   // GBK_TO_UNICODE[16971] := 16#7918;
   // GBK_TO_UNICODE[16972] := 16#B54B;
   // GBK_TO_UNICODE[16973] := 16#7919;
   // GBK_TO_UNICODE[16974] := 16#B54C;
   // GBK_TO_UNICODE[16975] := 16#791A;
   // GBK_TO_UNICODE[16976] := 16#B54D;
   // GBK_TO_UNICODE[16977] := 16#791B;
   // GBK_TO_UNICODE[16978] := 16#B54E;
   // GBK_TO_UNICODE[16979] := 16#791C;
   // GBK_TO_UNICODE[16980] := 16#B54F;
   // GBK_TO_UNICODE[16981] := 16#791D;
   // GBK_TO_UNICODE[16982] := 16#B550;
   // GBK_TO_UNICODE[16983] := 16#791F;
   // GBK_TO_UNICODE[16984] := 16#B551;
   // GBK_TO_UNICODE[16985] := 16#7920;
   // GBK_TO_UNICODE[16986] := 16#B552;
   // GBK_TO_UNICODE[16987] := 16#7921;
   // GBK_TO_UNICODE[16988] := 16#B553;
   // GBK_TO_UNICODE[16989] := 16#7922;
   // GBK_TO_UNICODE[16990] := 16#B554;
   // GBK_TO_UNICODE[16991] := 16#7923;
   // GBK_TO_UNICODE[16992] := 16#B555;
   // GBK_TO_UNICODE[16993] := 16#7925;
   // GBK_TO_UNICODE[16994] := 16#B556;
   // GBK_TO_UNICODE[16995] := 16#7926;
   // GBK_TO_UNICODE[16996] := 16#B557;
   // GBK_TO_UNICODE[16997] := 16#7927;
   // GBK_TO_UNICODE[16998] := 16#B558;
   // GBK_TO_UNICODE[16999] := 16#7928;
   // GBK_TO_UNICODE[17000] := 16#B559;
   // GBK_TO_UNICODE[17001] := 16#7929;
   // GBK_TO_UNICODE[17002] := 16#B55A;
   // GBK_TO_UNICODE[17003] := 16#792A;
   // GBK_TO_UNICODE[17004] := 16#B55B;
   // GBK_TO_UNICODE[17005] := 16#792B;
   // GBK_TO_UNICODE[17006] := 16#B55C;
   // GBK_TO_UNICODE[17007] := 16#792C;
   // GBK_TO_UNICODE[17008] := 16#B55D;
   // GBK_TO_UNICODE[17009] := 16#792D;
   // GBK_TO_UNICODE[17010] := 16#B55E;
   // GBK_TO_UNICODE[17011] := 16#792E;
   // GBK_TO_UNICODE[17012] := 16#B55F;
   // GBK_TO_UNICODE[17013] := 16#792F;
   // GBK_TO_UNICODE[17014] := 16#B560;
   // GBK_TO_UNICODE[17015] := 16#7930;
   // GBK_TO_UNICODE[17016] := 16#B561;
   // GBK_TO_UNICODE[17017] := 16#7931;
   // GBK_TO_UNICODE[17018] := 16#B562;
   // GBK_TO_UNICODE[17019] := 16#7932;
   // GBK_TO_UNICODE[17020] := 16#B563;
   // GBK_TO_UNICODE[17021] := 16#7933;
   // GBK_TO_UNICODE[17022] := 16#B564;
   // GBK_TO_UNICODE[17023] := 16#7935;
   // GBK_TO_UNICODE[17024] := 16#B565;
   // GBK_TO_UNICODE[17025] := 16#7936;
   // GBK_TO_UNICODE[17026] := 16#B566;
   // GBK_TO_UNICODE[17027] := 16#7937;
   // GBK_TO_UNICODE[17028] := 16#B567;
   // GBK_TO_UNICODE[17029] := 16#7938;
   // GBK_TO_UNICODE[17030] := 16#B568;
   // GBK_TO_UNICODE[17031] := 16#7939;
   // GBK_TO_UNICODE[17032] := 16#B569;
   // GBK_TO_UNICODE[17033] := 16#793D;
   // GBK_TO_UNICODE[17034] := 16#B56A;
   // GBK_TO_UNICODE[17035] := 16#793F;
   // GBK_TO_UNICODE[17036] := 16#B56B;
   // GBK_TO_UNICODE[17037] := 16#7942;
   // GBK_TO_UNICODE[17038] := 16#B56C;
   // GBK_TO_UNICODE[17039] := 16#7943;
   // GBK_TO_UNICODE[17040] := 16#B56D;
   // GBK_TO_UNICODE[17041] := 16#7944;
   // GBK_TO_UNICODE[17042] := 16#B56E;
   // GBK_TO_UNICODE[17043] := 16#7945;
   // GBK_TO_UNICODE[17044] := 16#B56F;
   // GBK_TO_UNICODE[17045] := 16#7947;
   // GBK_TO_UNICODE[17046] := 16#B570;
   // GBK_TO_UNICODE[17047] := 16#794A;
   // GBK_TO_UNICODE[17048] := 16#B571;
   // GBK_TO_UNICODE[17049] := 16#794B;
   // GBK_TO_UNICODE[17050] := 16#B572;
   // GBK_TO_UNICODE[17051] := 16#794C;
   // GBK_TO_UNICODE[17052] := 16#B573;
   // GBK_TO_UNICODE[17053] := 16#794D;
   // GBK_TO_UNICODE[17054] := 16#B574;
   // GBK_TO_UNICODE[17055] := 16#794E;
   // GBK_TO_UNICODE[17056] := 16#B575;
   // GBK_TO_UNICODE[17057] := 16#794F;
   // GBK_TO_UNICODE[17058] := 16#B576;
   // GBK_TO_UNICODE[17059] := 16#7950;
   // GBK_TO_UNICODE[17060] := 16#B577;
   // GBK_TO_UNICODE[17061] := 16#7951;
   // GBK_TO_UNICODE[17062] := 16#B578;
   // GBK_TO_UNICODE[17063] := 16#7952;
   // GBK_TO_UNICODE[17064] := 16#B579;
   // GBK_TO_UNICODE[17065] := 16#7954;
   // GBK_TO_UNICODE[17066] := 16#B57A;
   // GBK_TO_UNICODE[17067] := 16#7955;
